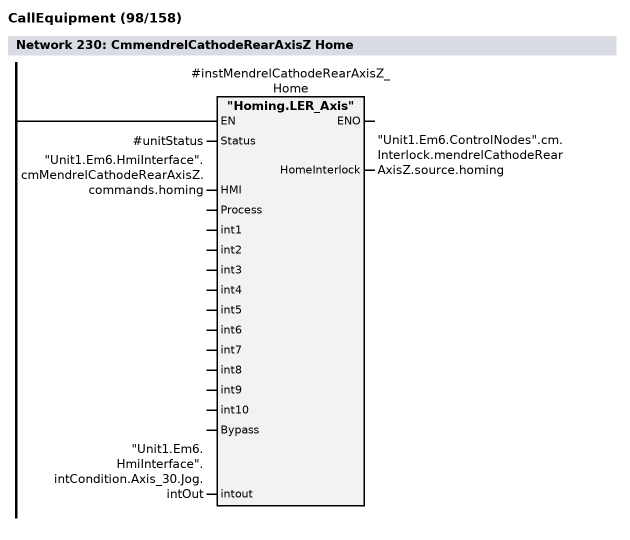
   RUNG wire#powerrail
      #instMendrelCathodeRearAxisZ_Home(Status := #unitStatus, HMI := "Unit1.Em6.HmiInterface".cmMendrelCathodeRearAxisZ.commands.homing, Process :=, int1 :=, int2 :=, int3 :=, int4 :=, int5 :=, int6 :=, int7 :=, int8 :=, int9 :=, int10 :=, Bypass :=, intout := "Unit1.Em6.HmiInterface".intCondition.Axis_30.Jog.intOut, HomeInterlock => "Unit1.Em6.ControlNodes".cm.Interlock.mendrelCathodeRearAxisZ.source.homing)
   END_RUNG
   // the same network as SCL:
   #instMendrelCathodeRearAxisZ_Home(Status := #unitStatus,   // "Homing.LER_Axis"
                           HMI := "Unit1.Em6.HmiInterface".cmMendrelCathodeRearAxisZ.commands.homing,
                           intout := "Unit1.Em6.HmiInterface".intCondition.Axis_30.Jog.intOut,
                           HomeInterlock => "Unit1.Em6.ControlNodes".cm.Interlock.mendrelCathodeRearAxisZ.source.homing);
END_REGION

REGION Network 231: CmmendrelCathodeRearAxisZ Position Absolute Jog
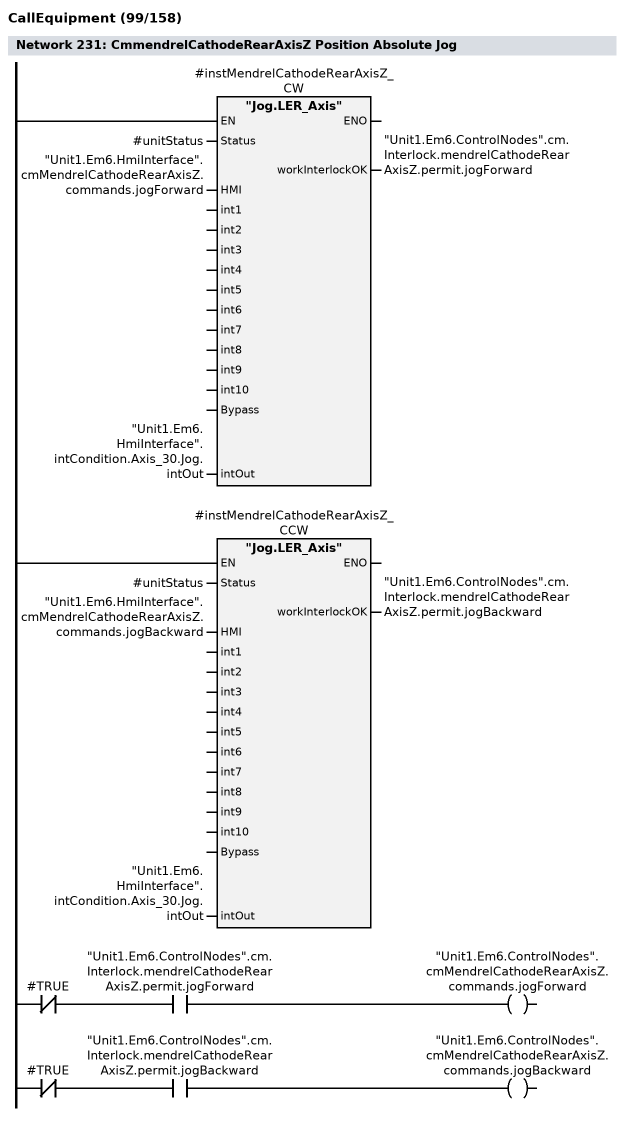
   RUNG wire#powerrail
      #instMendrelCathodeRearAxisZ_CW(Status := #unitStatus, HMI := "Unit1.Em6.HmiInterface".cmMendrelCathodeRearAxisZ.commands.jogForward, int1 :=, int2 :=, int3 :=, int4 :=, int5 :=, int6 :=, int7 :=, int8 :=, int9 :=, int10 :=, Bypass :=, intOut := "Unit1.Em6.HmiInterface".intCondition.Axis_30.Jog.intOut, workInterlockOK => "Unit1.Em6.ControlNodes".cm.Interlock.mendrelCathodeRearAxisZ.permit.jogForward)
   END_RUNG
   RUNG wire#powerrail
      #instMendrelCathodeRearAxisZ_CCW(Status := #unitStatus, HMI := "Unit1.Em6.HmiInterface".cmMendrelCathodeRearAxisZ.commands.jogBackward, int1 :=, int2 :=, int3 :=, int4 :=, int5 :=, int6 :=, int7 :=, int8 :=, int9 :=, int10 :=, Bypass :=, intOut := "Unit1.Em6.HmiInterface".intCondition.Axis_30.Jog.intOut, workInterlockOK => "Unit1.Em6.ControlNodes".cm.Interlock.mendrelCathodeRearAxisZ.permit.jogBackward)
   END_RUNG
   RUNG wire#powerrail
      I_Contact( #TRUE )
      Contact( "Unit1.Em6.ControlNodes".cm.Interlock.mendrelCathodeRearAxisZ.permit.jogForward )
      Coil( "Unit1.Em6.ControlNodes".cmMendrelCathodeRearAxisZ.commands.jogForward )
   END_RUNG
   RUNG wire#powerrail
      I_Contact( #TRUE )
      Contact( "Unit1.Em6.ControlNodes".cm.Interlock.mendrelCathodeRearAxisZ.permit.jogBackward )
      Coil( "Unit1.Em6.ControlNodes".cmMendrelCathodeRearAxisZ.commands.jogBackward )
   END_RUNG
   // the same network as SCL:
   #instMendrelCathodeRearAxisZ_CW(Status := #unitStatus,   // "Jog.LER_Axis"
                           HMI := "Unit1.Em6.HmiInterface".cmMendrelCathodeRearAxisZ.commands.jogForward,
                           intOut := "Unit1.Em6.HmiInterface".intCondition.Axis_30.Jog.intOut,
                           workInterlockOK => "Unit1.Em6.ControlNodes".cm.Interlock.mendrelCathodeRearAxisZ.permit.jogForward);
   #instMendrelCathodeRearAxisZ_CCW(Status := #unitStatus,   // "Jog.LER_Axis"
                           HMI := "Unit1.Em6.HmiInterface".cmMendrelCathodeRearAxisZ.commands.jogBackward,
                           intOut := "Unit1.Em6.HmiInterface".intCondition.Axis_30.Jog.intOut,
                           workInterlockOK => "Unit1.Em6.ControlNodes".cm.Interlock.mendrelCathodeRearAxisZ.permit.jogBackward);
   "Unit1.Em6.ControlNodes".cmMendrelCathodeRearAxisZ.commands.jogForward := NOT #TRUE AND "Unit1.Em6.ControlNodes".cm.Interlock.mendrelCathodeRearAxisZ.permit.jogForward;
   "Unit1.Em6.ControlNodes".cmMendrelCathodeRearAxisZ.commands.jogBackward := NOT #TRUE AND "Unit1.Em6.ControlNodes".cm.Interlock.mendrelCathodeRearAxisZ.permit.jogBackward;
END_REGION

REGION Network 232: CmmendrelCathodeRearAxisZ Position Absolute Position0
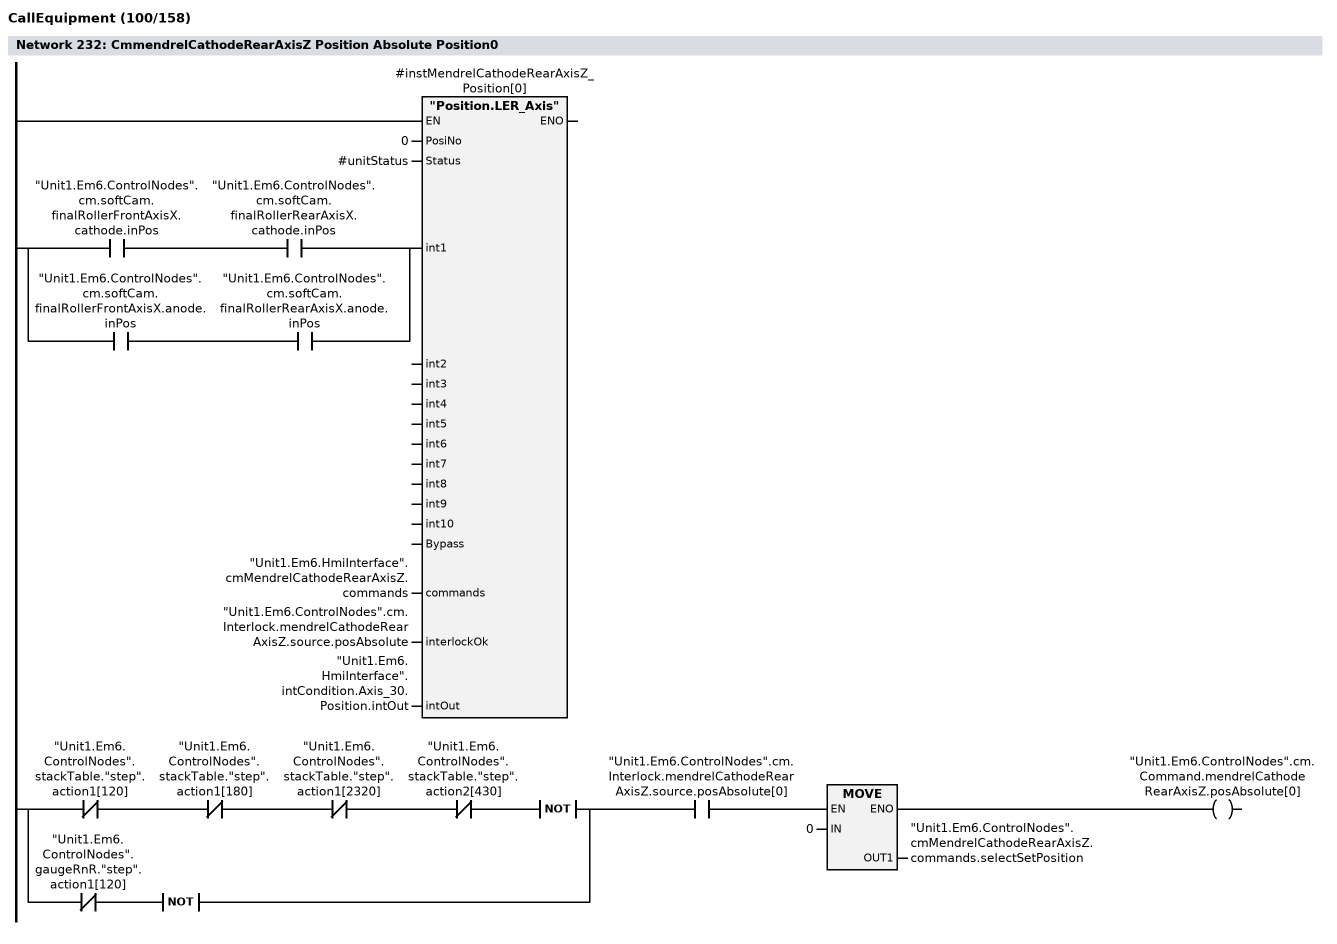
   RUNG wire#powerrail
      #instMendrelCathodeRearAxisZ_Position[0](int1 := wire#w1, PosiNo := 0, Status := #unitStatus, int2 :=, int3 :=, int4 :=, int5 :=, int6 :=, int7 :=, int8 :=, int9 :=, int10 :=, Bypass :=, commands := "Unit1.Em6.HmiInterface".cmMendrelCathodeRearAxisZ.commands, interlockOk := "Unit1.Em6.ControlNodes".cm.Interlock.mendrelCathodeRearAxisZ.source.posAbsolute, intOut := "Unit1.Em6.HmiInterface".intCondition.Axis_30.Position.intOut)
   END_RUNG
   RUNG wire#powerrail
      Contact( "Unit1.Em6.ControlNodes".cm.softCam.finalRollerFrontAxisX.cathode.inPos )
      Contact( "Unit1.Em6.ControlNodes".cm.softCam.finalRollerRearAxisX.cathode.inPos )
   END_RUNG wire#w1
   RUNG wire#powerrail
      Contact( "Unit1.Em6.ControlNodes".cm.softCam.finalRollerFrontAxisX.anode.inPos )
      Contact( "Unit1.Em6.ControlNodes".cm.softCam.finalRollerRearAxisX.anode.inPos )
   END_RUNG wire#w1
   RUNG wire#powerrail
      I_Contact( "Unit1.Em6.ControlNodes".stackTable."step".action1[120] )
      I_Contact( "Unit1.Em6.ControlNodes".stackTable."step".action1[180] )
      I_Contact( "Unit1.Em6.ControlNodes".stackTable."step".action1[2320] )
      I_Contact( "Unit1.Em6.ControlNodes".stackTable."step".action2[430] )
      Not()
      wire#w2
      Contact( "Unit1.Em6.ControlNodes".cm.Interlock.mendrelCathodeRearAxisZ.source.posAbsolute[0] )
      Move(in := 0, out1 => "Unit1.Em6.ControlNodes".cmMendrelCathodeRearAxisZ.commands.selectSetPosition)
      Coil( "Unit1.Em6.ControlNodes".cm.Command.mendrelCathodeRearAxisZ.posAbsolute[0] )
   END_RUNG
   RUNG wire#powerrail
      I_Contact( "Unit1.Em6.ControlNodes".gaugeRnR."step".action1[120] )
      Not()
   END_RUNG wire#w2
   // the same network as SCL:
   #instMendrelCathodeRearAxisZ_Position[0](PosiNo := 0,   // "Position.LER_Axis"
                           Status := #unitStatus,
                           int1 := ("Unit1.Em6.ControlNodes".cm.softCam.finalRollerFrontAxisX.cathode.inPos AND "Unit1.Em6.ControlNodes".cm.softCam.finalRollerRearAxisX.cathode.inPos) OR ("Unit1.Em6.ControlNodes".cm.softCam.finalRollerFrontAxisX.anode.inPos AND "Unit1.Em6.ControlNodes".cm.softCam.finalRollerRearAxisX.anode.inPos),
                           commands := "Unit1.Em6.HmiInterface".cmMendrelCathodeRearAxisZ.commands,
                           interlockOk := "Unit1.Em6.ControlNodes".cm.Interlock.mendrelCathodeRearAxisZ.source.posAbsolute,
                           intOut := "Unit1.Em6.HmiInterface".intCondition.Axis_30.Position.intOut);
   #_w1 := (NOT (NOT "Unit1.Em6.ControlNodes".stackTable."step".action1[120] AND NOT "Unit1.Em6.ControlNodes".stackTable."step".action1[180] AND NOT "Unit1.Em6.ControlNodes".stackTable."step".action1[2320] AND NOT "Unit1.Em6.ControlNodes".stackTable."step".action2[430]) OR NOT (NOT "Unit1.Em6.ControlNodes".gaugeRnR."step".action1[120])) AND "Unit1.Em6.ControlNodes".cm.Interlock.mendrelCathodeRearAxisZ.source.posAbsolute[0];
   IF #_w1 THEN "Unit1.Em6.ControlNodes".cmMendrelCathodeRearAxisZ.commands.selectSetPosition := 0; END_IF;
   "Unit1.Em6.ControlNodes".cm.Command.mendrelCathodeRearAxisZ.posAbsolute[0] := #_w1;
END_REGION

REGION Network 233: CmmendrelCathodeRearAxisZ Position Absolute Position1
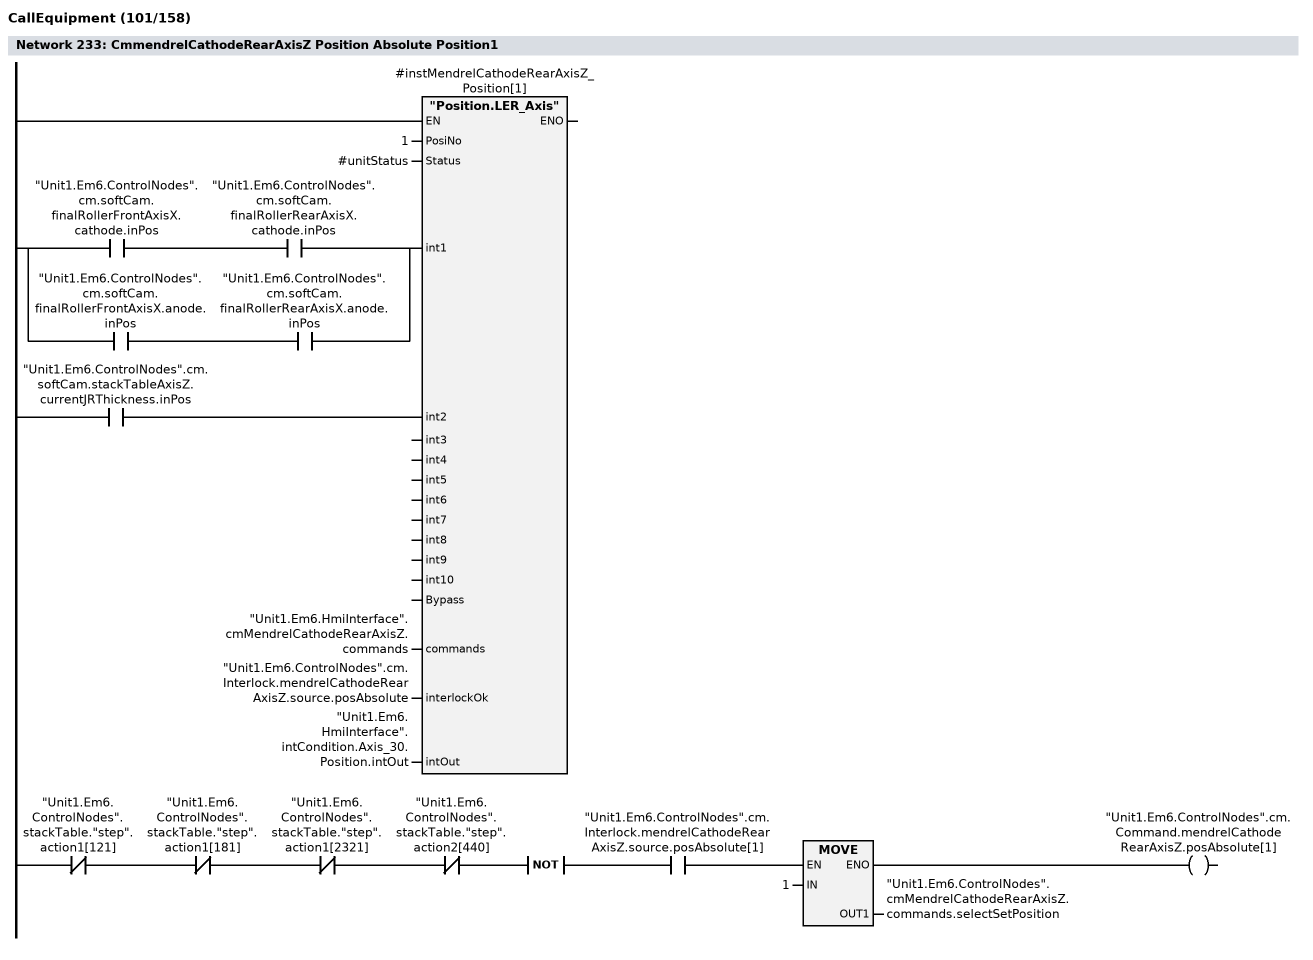
   RUNG wire#powerrail
      #instMendrelCathodeRearAxisZ_Position[1](int1 := wire#w1, int2 := wire#w2, PosiNo := 1, Status := #unitStatus, int3 :=, int4 :=, int5 :=, int6 :=, int7 :=, int8 :=, int9 :=, int10 :=, Bypass :=, commands := "Unit1.Em6.HmiInterface".cmMendrelCathodeRearAxisZ.commands, interlockOk := "Unit1.Em6.ControlNodes".cm.Interlock.mendrelCathodeRearAxisZ.source.posAbsolute, intOut := "Unit1.Em6.HmiInterface".intCondition.Axis_30.Position.intOut)
   END_RUNG
   RUNG wire#powerrail
      Contact( "Unit1.Em6.ControlNodes".cm.softCam.finalRollerFrontAxisX.cathode.inPos )
      Contact( "Unit1.Em6.ControlNodes".cm.softCam.finalRollerRearAxisX.cathode.inPos )
   END_RUNG wire#w1
   RUNG wire#powerrail
      Contact( "Unit1.Em6.ControlNodes".cm.softCam.finalRollerFrontAxisX.anode.inPos )
      Contact( "Unit1.Em6.ControlNodes".cm.softCam.finalRollerRearAxisX.anode.inPos )
   END_RUNG wire#w1
   RUNG wire#powerrail
      Contact( "Unit1.Em6.ControlNodes".cm.softCam.stackTableAxisZ.currentJRThickness.inPos )
   END_RUNG wire#w2
   RUNG wire#powerrail
      I_Contact( "Unit1.Em6.ControlNodes".stackTable."step".action1[121] )
      I_Contact( "Unit1.Em6.ControlNodes".stackTable."step".action1[181] )
      I_Contact( "Unit1.Em6.ControlNodes".stackTable."step".action1[2321] )
      I_Contact( "Unit1.Em6.ControlNodes".stackTable."step".action2[440] )
      Not()
      Contact( "Unit1.Em6.ControlNodes".cm.Interlock.mendrelCathodeRearAxisZ.source.posAbsolute[1] )
      Move(in := 1, out1 => "Unit1.Em6.ControlNodes".cmMendrelCathodeRearAxisZ.commands.selectSetPosition)
      Coil( "Unit1.Em6.ControlNodes".cm.Command.mendrelCathodeRearAxisZ.posAbsolute[1] )
   END_RUNG
   // the same network as SCL:
   #instMendrelCathodeRearAxisZ_Position[1](PosiNo := 1,   // "Position.LER_Axis"
                           Status := #unitStatus,
                           int1 := ("Unit1.Em6.ControlNodes".cm.softCam.finalRollerFrontAxisX.cathode.inPos AND "Unit1.Em6.ControlNodes".cm.softCam.finalRollerRearAxisX.cathode.inPos) OR ("Unit1.Em6.ControlNodes".cm.softCam.finalRollerFrontAxisX.anode.inPos AND "Unit1.Em6.ControlNodes".cm.softCam.finalRollerRearAxisX.anode.inPos),
                           int2 := "Unit1.Em6.ControlNodes".cm.softCam.stackTableAxisZ.currentJRThickness.inPos,
                           commands := "Unit1.Em6.HmiInterface".cmMendrelCathodeRearAxisZ.commands,
                           interlockOk := "Unit1.Em6.ControlNodes".cm.Interlock.mendrelCathodeRearAxisZ.source.posAbsolute,
                           intOut := "Unit1.Em6.HmiInterface".intCondition.Axis_30.Position.intOut);
   #_w1 := NOT (NOT "Unit1.Em6.ControlNodes".stackTable."step".action1[121] AND NOT "Unit1.Em6.ControlNodes".stackTable."step".action1[181] AND NOT "Unit1.Em6.ControlNodes".stackTable."step".action1[2321] AND NOT "Unit1.Em6.ControlNodes".stackTable."step".action2[440]) AND "Unit1.Em6.ControlNodes".cm.Interlock.mendrelCathodeRearAxisZ.source.posAbsolute[1];
   IF #_w1 THEN "Unit1.Em6.ControlNodes".cmMendrelCathodeRearAxisZ.commands.selectSetPosition := 1; END_IF;
   "Unit1.Em6.ControlNodes".cm.Command.mendrelCathodeRearAxisZ.posAbsolute[1] := #_w1;
END_REGION

REGION Network 234: CmmendrelCathodeRearAxisZ Position Absolute Position2
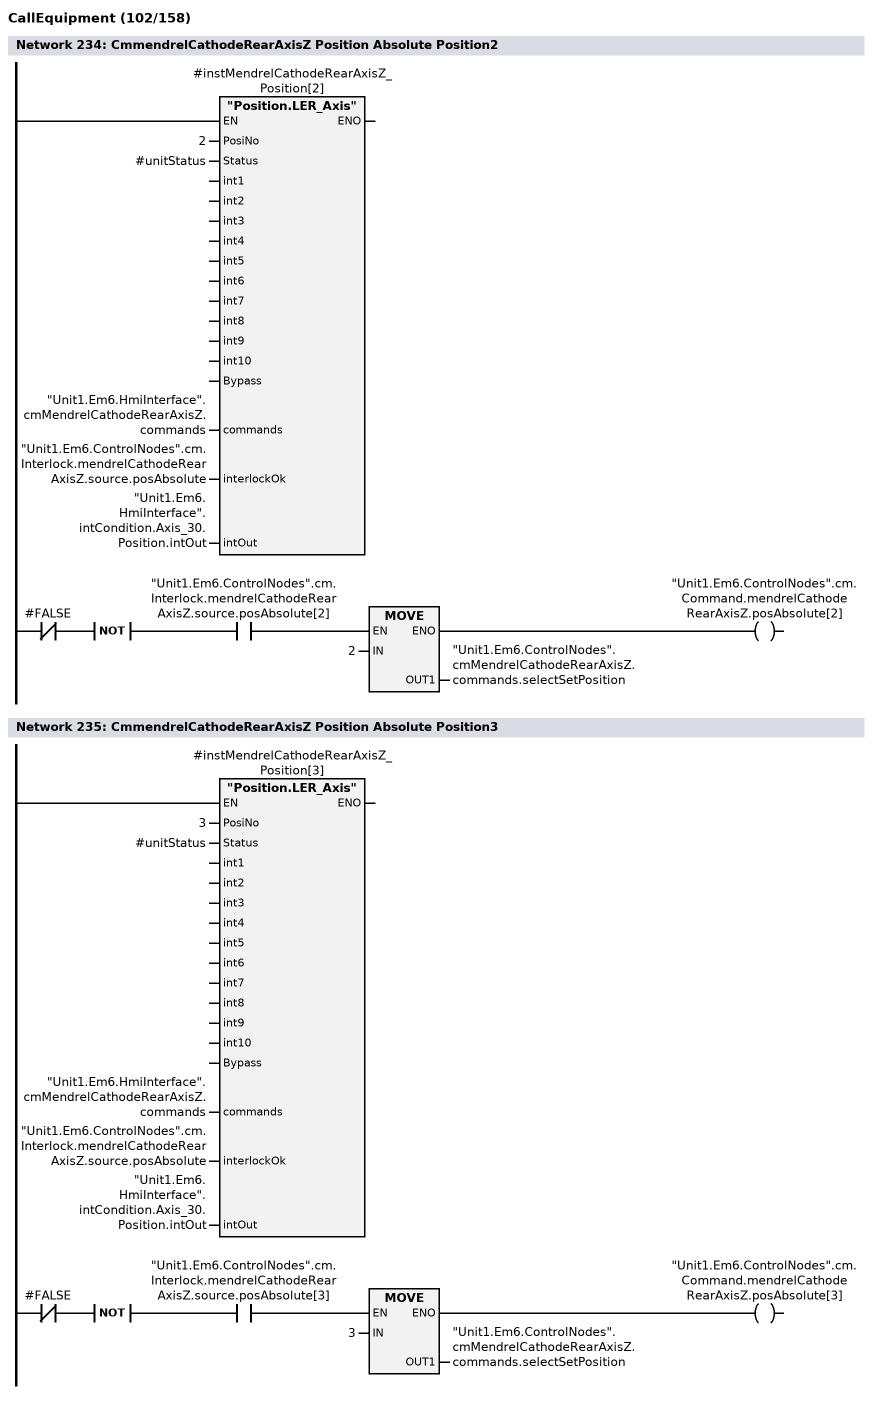
   RUNG wire#powerrail
      #instMendrelCathodeRearAxisZ_Position[2](PosiNo := 2, Status := #unitStatus, int1 :=, int2 :=, int3 :=, int4 :=, int5 :=, int6 :=, int7 :=, int8 :=, int9 :=, int10 :=, Bypass :=, commands := "Unit1.Em6.HmiInterface".cmMendrelCathodeRearAxisZ.commands, interlockOk := "Unit1.Em6.ControlNodes".cm.Interlock.mendrelCathodeRearAxisZ.source.posAbsolute, intOut := "Unit1.Em6.HmiInterface".intCondition.Axis_30.Position.intOut)
   END_RUNG
   RUNG wire#powerrail
      I_Contact( #FALSE )
      Not()
      Contact( "Unit1.Em6.ControlNodes".cm.Interlock.mendrelCathodeRearAxisZ.source.posAbsolute[2] )
      Move(in := 2, out1 => "Unit1.Em6.ControlNodes".cmMendrelCathodeRearAxisZ.commands.selectSetPosition)
      Coil( "Unit1.Em6.ControlNodes".cm.Command.mendrelCathodeRearAxisZ.posAbsolute[2] )
   END_RUNG
   // the same network as SCL:
   #instMendrelCathodeRearAxisZ_Position[2](PosiNo := 2,   // "Position.LER_Axis"
                           Status := #unitStatus,
                           commands := "Unit1.Em6.HmiInterface".cmMendrelCathodeRearAxisZ.commands,
                           interlockOk := "Unit1.Em6.ControlNodes".cm.Interlock.mendrelCathodeRearAxisZ.source.posAbsolute,
                           intOut := "Unit1.Em6.HmiInterface".intCondition.Axis_30.Position.intOut);
   #_w1 := NOT (NOT #FALSE) AND "Unit1.Em6.ControlNodes".cm.Interlock.mendrelCathodeRearAxisZ.source.posAbsolute[2];
   IF #_w1 THEN "Unit1.Em6.ControlNodes".cmMendrelCathodeRearAxisZ.commands.selectSetPosition := 2; END_IF;
   "Unit1.Em6.ControlNodes".cm.Command.mendrelCathodeRearAxisZ.posAbsolute[2] := #_w1;
END_REGION

REGION Network 235: CmmendrelCathodeRearAxisZ Position Absolute Position3
   RUNG wire#powerrail
      #instMendrelCathodeRearAxisZ_Position[3](PosiNo := 3, Status := #unitStatus, int1 :=, int2 :=, int3 :=, int4 :=, int5 :=, int6 :=, int7 :=, int8 :=, int9 :=, int10 :=, Bypass :=, commands := "Unit1.Em6.HmiInterface".cmMendrelCathodeRearAxisZ.commands, interlockOk := "Unit1.Em6.ControlNodes".cm.Interlock.mendrelCathodeRearAxisZ.source.posAbsolute, intOut := "Unit1.Em6.HmiInterface".intCondition.Axis_30.Position.intOut)
   END_RUNG
   RUNG wire#powerrail
      I_Contact( #FALSE )
      Not()
      Contact( "Unit1.Em6.ControlNodes".cm.Interlock.mendrelCathodeRearAxisZ.source.posAbsolute[3] )
      Move(in := 3, out1 => "Unit1.Em6.ControlNodes".cmMendrelCathodeRearAxisZ.commands.selectSetPosition)
      Coil( "Unit1.Em6.ControlNodes".cm.Command.mendrelCathodeRearAxisZ.posAbsolute[3] )
   END_RUNG
   // the same network as SCL:
   #instMendrelCathodeRearAxisZ_Position[3](PosiNo := 3,   // "Position.LER_Axis"
                           Status := #unitStatus,
                           commands := "Unit1.Em6.HmiInterface".cmMendrelCathodeRearAxisZ.commands,
                           interlockOk := "Unit1.Em6.ControlNodes".cm.Interlock.mendrelCathodeRearAxisZ.source.posAbsolute,
                           intOut := "Unit1.Em6.HmiInterface".intCondition.Axis_30.Position.intOut);
   #_w1 := NOT (NOT #FALSE) AND "Unit1.Em6.ControlNodes".cm.Interlock.mendrelCathodeRearAxisZ.source.posAbsolute[3];
   IF #_w1 THEN "Unit1.Em6.ControlNodes".cmMendrelCathodeRearAxisZ.commands.selectSetPosition := 3; END_IF;
   "Unit1.Em6.ControlNodes".cm.Command.mendrelCathodeRearAxisZ.posAbsolute[3] := #_w1;
END_REGION

REGION Network 236: CmmendrelCathodeRearAxisZ Position Absolute Position4
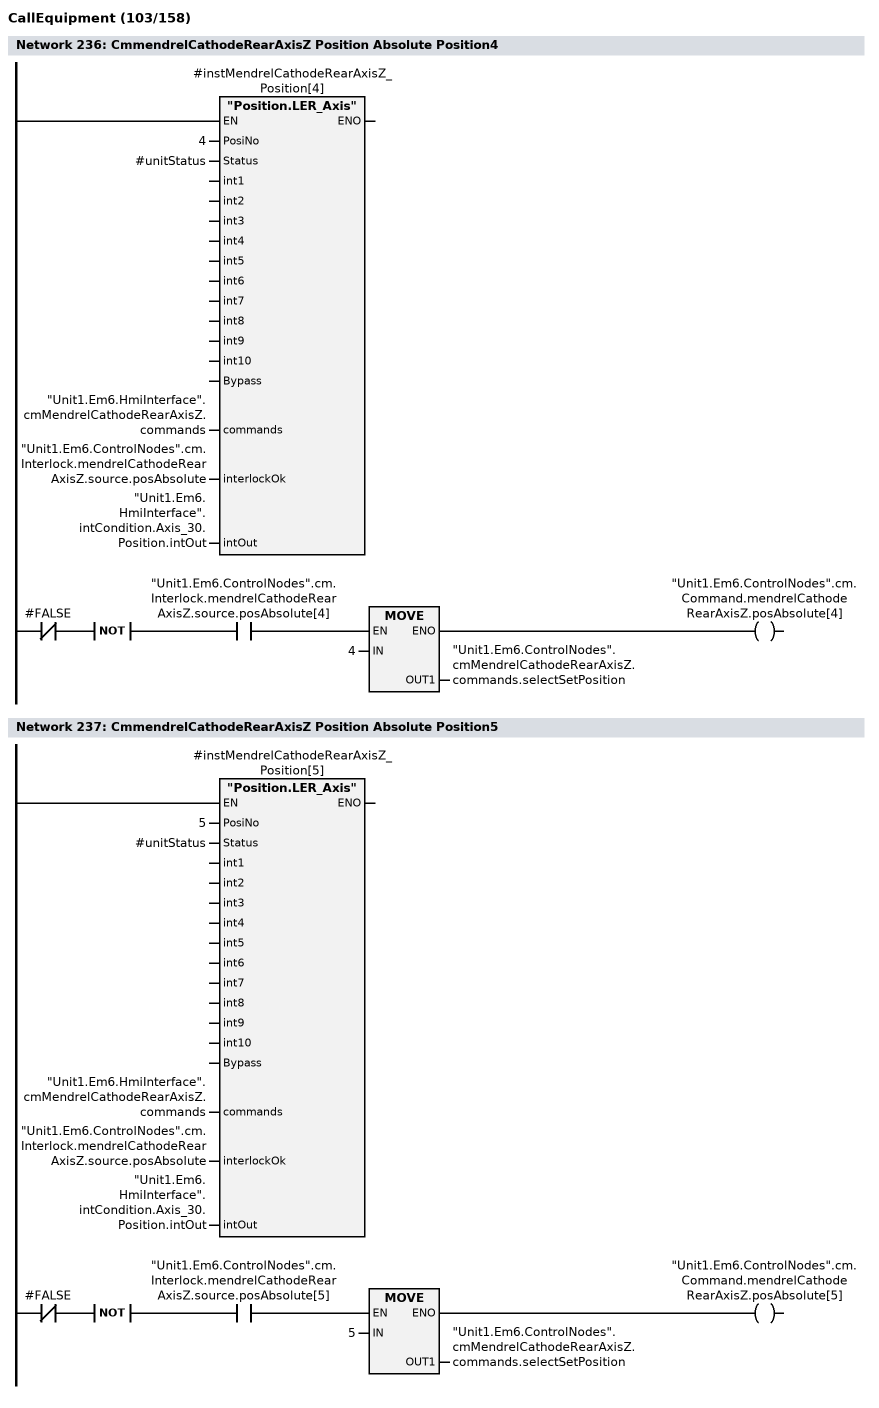
   RUNG wire#powerrail
      #instMendrelCathodeRearAxisZ_Position[4](PosiNo := 4, Status := #unitStatus, int1 :=, int2 :=, int3 :=, int4 :=, int5 :=, int6 :=, int7 :=, int8 :=, int9 :=, int10 :=, Bypass :=, commands := "Unit1.Em6.HmiInterface".cmMendrelCathodeRearAxisZ.commands, interlockOk := "Unit1.Em6.ControlNodes".cm.Interlock.mendrelCathodeRearAxisZ.source.posAbsolute, intOut := "Unit1.Em6.HmiInterface".intCondition.Axis_30.Position.intOut)
   END_RUNG
   RUNG wire#powerrail
      I_Contact( #FALSE )
      Not()
      Contact( "Unit1.Em6.ControlNodes".cm.Interlock.mendrelCathodeRearAxisZ.source.posAbsolute[4] )
      Move(in := 4, out1 => "Unit1.Em6.ControlNodes".cmMendrelCathodeRearAxisZ.commands.selectSetPosition)
      Coil( "Unit1.Em6.ControlNodes".cm.Command.mendrelCathodeRearAxisZ.posAbsolute[4] )
   END_RUNG
   // the same network as SCL:
   #instMendrelCathodeRearAxisZ_Position[4](PosiNo := 4,   // "Position.LER_Axis"
                           Status := #unitStatus,
                           commands := "Unit1.Em6.HmiInterface".cmMendrelCathodeRearAxisZ.commands,
                           interlockOk := "Unit1.Em6.ControlNodes".cm.Interlock.mendrelCathodeRearAxisZ.source.posAbsolute,
                           intOut := "Unit1.Em6.HmiInterface".intCondition.Axis_30.Position.intOut);
   #_w1 := NOT (NOT #FALSE) AND "Unit1.Em6.ControlNodes".cm.Interlock.mendrelCathodeRearAxisZ.source.posAbsolute[4];
   IF #_w1 THEN "Unit1.Em6.ControlNodes".cmMendrelCathodeRearAxisZ.commands.selectSetPosition := 4; END_IF;
   "Unit1.Em6.ControlNodes".cm.Command.mendrelCathodeRearAxisZ.posAbsolute[4] := #_w1;
END_REGION

REGION Network 237: CmmendrelCathodeRearAxisZ Position Absolute Position5
   RUNG wire#powerrail
      #instMendrelCathodeRearAxisZ_Position[5](PosiNo := 5, Status := #unitStatus, int1 :=, int2 :=, int3 :=, int4 :=, int5 :=, int6 :=, int7 :=, int8 :=, int9 :=, int10 :=, Bypass :=, commands := "Unit1.Em6.HmiInterface".cmMendrelCathodeRearAxisZ.commands, interlockOk := "Unit1.Em6.ControlNodes".cm.Interlock.mendrelCathodeRearAxisZ.source.posAbsolute, intOut := "Unit1.Em6.HmiInterface".intCondition.Axis_30.Position.intOut)
   END_RUNG
   RUNG wire#powerrail
      I_Contact( #FALSE )
      Not()
      Contact( "Unit1.Em6.ControlNodes".cm.Interlock.mendrelCathodeRearAxisZ.source.posAbsolute[5] )
      Move(in := 5, out1 => "Unit1.Em6.ControlNodes".cmMendrelCathodeRearAxisZ.commands.selectSetPosition)
      Coil( "Unit1.Em6.ControlNodes".cm.Command.mendrelCathodeRearAxisZ.posAbsolute[5] )
   END_RUNG
   // the same network as SCL:
   #instMendrelCathodeRearAxisZ_Position[5](PosiNo := 5,   // "Position.LER_Axis"
                           Status := #unitStatus,
                           commands := "Unit1.Em6.HmiInterface".cmMendrelCathodeRearAxisZ.commands,
                           interlockOk := "Unit1.Em6.ControlNodes".cm.Interlock.mendrelCathodeRearAxisZ.source.posAbsolute,
                           intOut := "Unit1.Em6.HmiInterface".intCondition.Axis_30.Position.intOut);
   #_w1 := NOT (NOT #FALSE) AND "Unit1.Em6.ControlNodes".cm.Interlock.mendrelCathodeRearAxisZ.source.posAbsolute[5];
   IF #_w1 THEN "Unit1.Em6.ControlNodes".cmMendrelCathodeRearAxisZ.commands.selectSetPosition := 5; END_IF;
   "Unit1.Em6.ControlNodes".cm.Command.mendrelCathodeRearAxisZ.posAbsolute[5] := #_w1;
END_REGION

REGION Network 238: CmmendrelCathodeRearAxisZ Summary Command
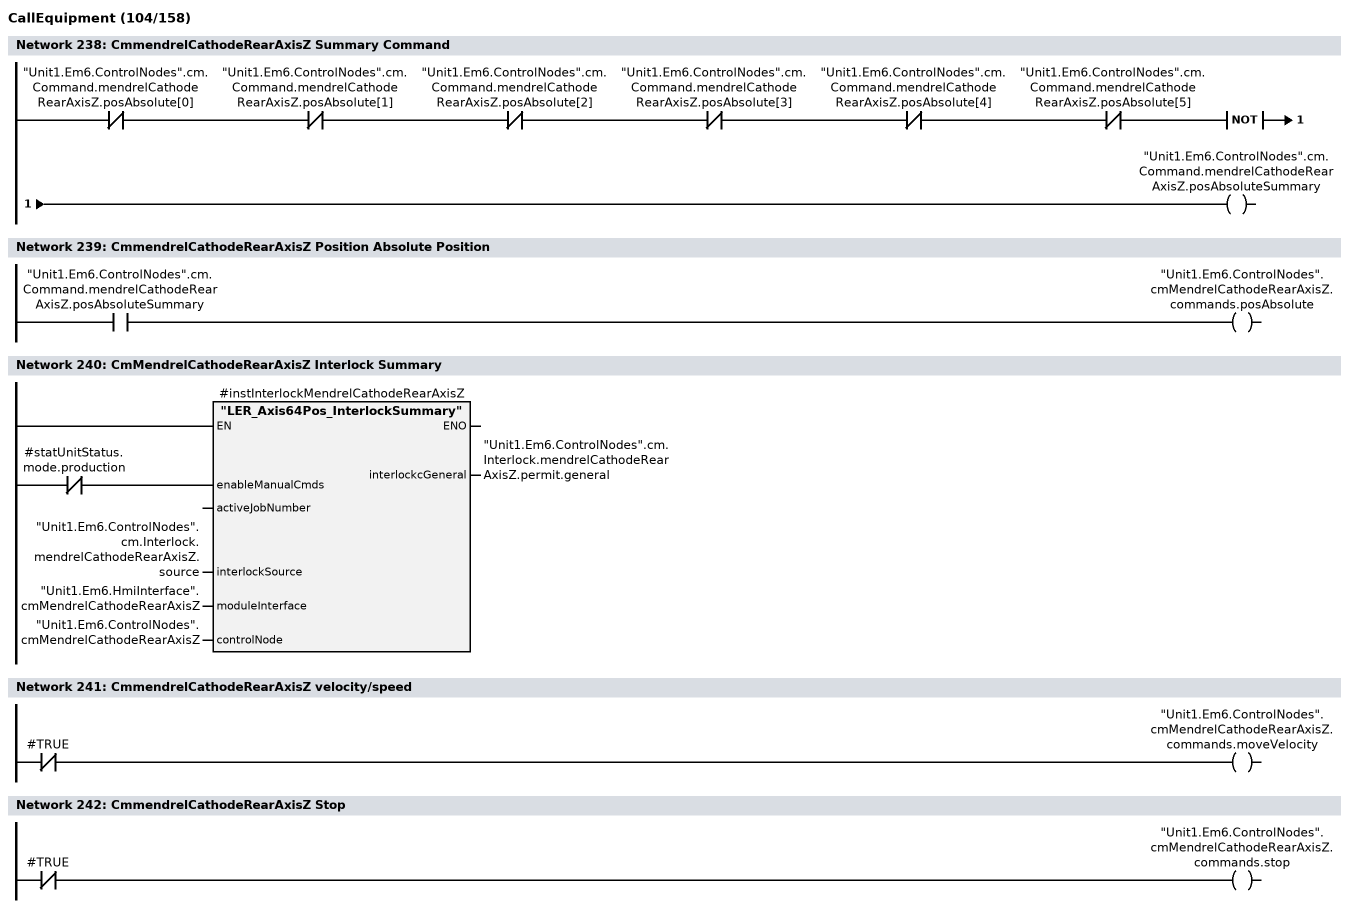
   RUNG wire#powerrail
      I_Contact( "Unit1.Em6.ControlNodes".cm.Command.mendrelCathodeRearAxisZ.posAbsolute[0] )
      I_Contact( "Unit1.Em6.ControlNodes".cm.Command.mendrelCathodeRearAxisZ.posAbsolute[1] )
      I_Contact( "Unit1.Em6.ControlNodes".cm.Command.mendrelCathodeRearAxisZ.posAbsolute[2] )
      I_Contact( "Unit1.Em6.ControlNodes".cm.Command.mendrelCathodeRearAxisZ.posAbsolute[3] )
      I_Contact( "Unit1.Em6.ControlNodes".cm.Command.mendrelCathodeRearAxisZ.posAbsolute[4] )
      I_Contact( "Unit1.Em6.ControlNodes".cm.Command.mendrelCathodeRearAxisZ.posAbsolute[5] )
      Not()
      Coil( "Unit1.Em6.ControlNodes".cm.Command.mendrelCathodeRearAxisZ.posAbsoluteSummary )
   END_RUNG
   // the same network as SCL:
   "Unit1.Em6.ControlNodes".cm.Command.mendrelCathodeRearAxisZ.posAbsoluteSummary := NOT (NOT "Unit1.Em6.ControlNodes".cm.Command.mendrelCathodeRearAxisZ.posAbsolute[0] AND NOT "Unit1.Em6.ControlNodes".cm.Command.mendrelCathodeRearAxisZ.posAbsolute[1] AND NOT "Unit1.Em6.ControlNodes".cm.Command.mendrelCathodeRearAxisZ.posAbsolute[2] AND NOT "Unit1.Em6.ControlNodes".cm.Command.mendrelCathodeRearAxisZ.posAbsolute[3] AND NOT "Unit1.Em6.ControlNodes".cm.Command.mendrelCathodeRearAxisZ.posAbsolute[4] AND NOT "Unit1.Em6.ControlNodes".cm.Command.mendrelCathodeRearAxisZ.posAbsolute[5]);
END_REGION

REGION Network 239: CmmendrelCathodeRearAxisZ Position Absolute Position
   RUNG wire#powerrail
      Contact( "Unit1.Em6.ControlNodes".cm.Command.mendrelCathodeRearAxisZ.posAbsoluteSummary )
      Coil( "Unit1.Em6.ControlNodes".cmMendrelCathodeRearAxisZ.commands.posAbsolute )
   END_RUNG
   // the same network as SCL:
   "Unit1.Em6.ControlNodes".cmMendrelCathodeRearAxisZ.commands.posAbsolute := "Unit1.Em6.ControlNodes".cm.Command.mendrelCathodeRearAxisZ.posAbsoluteSummary;
END_REGION

REGION Network 240: CmMendrelCathodeRearAxisZ Interlock Summary
   RUNG wire#powerrail
      #instInterlockMendrelCathodeRearAxisZ(enableManualCmds := wire#w1, activeJobNumber :=, interlockSource := "Unit1.Em6.ControlNodes".cm.Interlock.mendrelCathodeRearAxisZ.source, moduleInterface := "Unit1.Em6.HmiInterface".cmMendrelCathodeRearAxisZ, controlNode := "Unit1.Em6.ControlNodes".cmMendrelCathodeRearAxisZ, interlockcGeneral => "Unit1.Em6.ControlNodes".cm.Interlock.mendrelCathodeRearAxisZ.permit.general)
   END_RUNG
   RUNG wire#powerrail
      I_Contact( #statUnitStatus.mode.production )
   END_RUNG wire#w1
   // the same network as SCL:
   #instInterlockMendrelCathodeRearAxisZ(enableManualCmds := NOT #statUnitStatus.mode.production,   // "LER_Axis64Pos_InterlockSummary"
                           interlockSource := "Unit1.Em6.ControlNodes".cm.Interlock.mendrelCathodeRearAxisZ.source,
                           moduleInterface := "Unit1.Em6.HmiInterface".cmMendrelCathodeRearAxisZ,
                           controlNode := "Unit1.Em6.ControlNodes".cmMendrelCathodeRearAxisZ,
                           interlockcGeneral => "Unit1.Em6.ControlNodes".cm.Interlock.mendrelCathodeRearAxisZ.permit.general);
END_REGION

REGION Network 241: CmmendrelCathodeRearAxisZ velocity/speed
   RUNG wire#powerrail
      I_Contact( #TRUE )
      Coil( "Unit1.Em6.ControlNodes".cmMendrelCathodeRearAxisZ.commands.moveVelocity )
   END_RUNG
   // the same network as SCL:
   "Unit1.Em6.ControlNodes".cmMendrelCathodeRearAxisZ.commands.moveVelocity := NOT #TRUE;
END_REGION

REGION Network 242: CmmendrelCathodeRearAxisZ Stop
   RUNG wire#powerrail
      I_Contact( #TRUE )
      Coil( "Unit1.Em6.ControlNodes".cmMendrelCathodeRearAxisZ.commands.stop )
   END_RUNG
   // the same network as SCL:
   "Unit1.Em6.ControlNodes".cmMendrelCathodeRearAxisZ.commands.stop := NOT #TRUE;
END_REGION

REGION Network 243: Call CM Cathode Mandrel Rear Z-Axis (LBC_Axis64Pos)
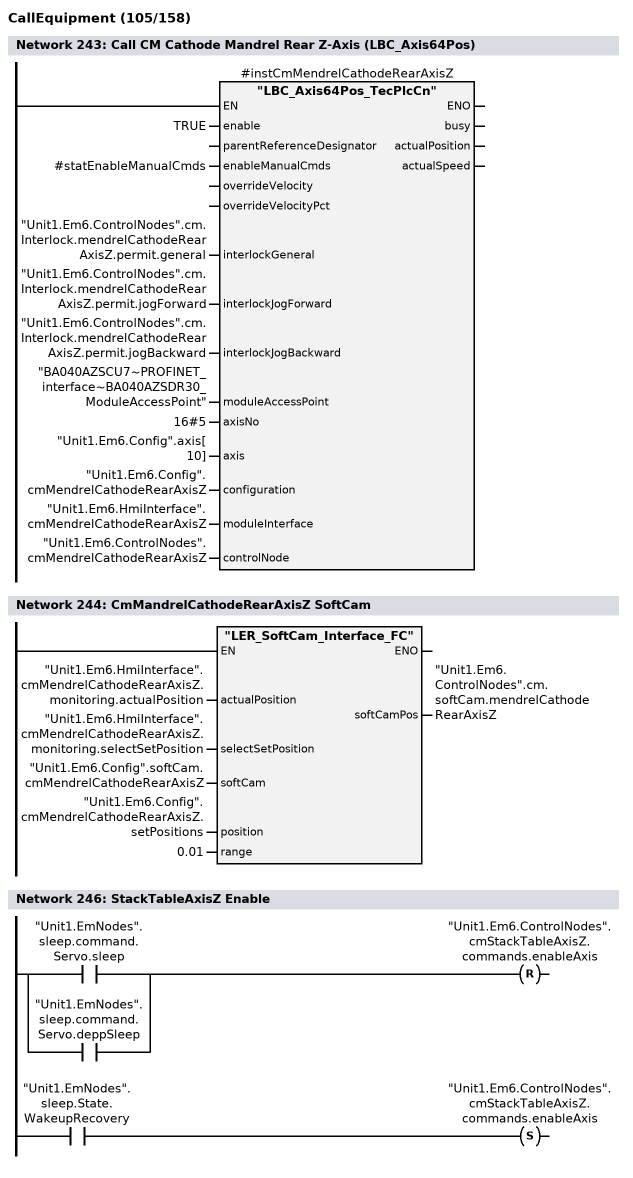
   RUNG wire#powerrail
      #instCmMendrelCathodeRearAxisZ(enable := TRUE, parentReferenceDesignator :=, enableManualCmds := #statEnableManualCmds, overrideVelocity :=, overrideVelocityPct :=, interlockGeneral := "Unit1.Em6.ControlNodes".cm.Interlock.mendrelCathodeRearAxisZ.permit.general, interlockJogForward := "Unit1.Em6.ControlNodes".cm.Interlock.mendrelCathodeRearAxisZ.permit.jogForward, interlockJogBackward := "Unit1.Em6.ControlNodes".cm.Interlock.mendrelCathodeRearAxisZ.permit.jogBackward, moduleAccessPoint := "BA040AZSCU7~PROFINET_interface~BA040AZSDR30_ModuleAccessPoint", axisNo := 16#5, axis := "Unit1.Em6.Config".axis[10], configuration := "Unit1.Em6.Config".cmMendrelCathodeRearAxisZ, moduleInterface := "Unit1.Em6.HmiInterface".cmMendrelCathodeRearAxisZ, controlNode := "Unit1.Em6.ControlNodes".cmMendrelCathodeRearAxisZ, busy =>, actualPosition =>, actualSpeed =>)
   END_RUNG
   // the same network as SCL:
   #instCmMendrelCathodeRearAxisZ(enable := TRUE,   // "LBC_Axis64Pos_TecPlcCn"
                           enableManualCmds := #statEnableManualCmds,
                           interlockGeneral := "Unit1.Em6.ControlNodes".cm.Interlock.mendrelCathodeRearAxisZ.permit.general,
                           interlockJogForward := "Unit1.Em6.ControlNodes".cm.Interlock.mendrelCathodeRearAxisZ.permit.jogForward,
                           interlockJogBackward := "Unit1.Em6.ControlNodes".cm.Interlock.mendrelCathodeRearAxisZ.permit.jogBackward,
                           moduleAccessPoint := "BA040AZSCU7~PROFINET_interface~BA040AZSDR30_ModuleAccessPoint",
                           axisNo := 16#5,
                           axis := "Unit1.Em6.Config".axis[10],
                           configuration := "Unit1.Em6.Config".cmMendrelCathodeRearAxisZ,
                           moduleInterface := "Unit1.Em6.HmiInterface".cmMendrelCathodeRearAxisZ,
                           controlNode := "Unit1.Em6.ControlNodes".cmMendrelCathodeRearAxisZ);
END_REGION

REGION Network 244: CmMandrelCathodeRearAxisZ SoftCam
   RUNG wire#powerrail
      "LER_SoftCam_Interface_FC"(actualPosition := "Unit1.Em6.HmiInterface".cmMendrelCathodeRearAxisZ.monitoring.actualPosition, selectSetPosition := "Unit1.Em6.HmiInterface".cmMendrelCathodeRearAxisZ.monitoring.selectSetPosition, softCam := "Unit1.Em6.Config".softCam.cmMendrelCathodeRearAxisZ, position := "Unit1.Em6.Config".cmMendrelCathodeRearAxisZ.setPositions, range := 0.01, softCamPos => "Unit1.Em6.ControlNodes".cm.softCam.mendrelCathodeRearAxisZ)
   END_RUNG
   // the same network as SCL:
   "LER_SoftCam_Interface_FC"(actualPosition := "Unit1.Em6.HmiInterface".cmMendrelCathodeRearAxisZ.monitoring.actualPosition,
                           selectSetPosition := "Unit1.Em6.HmiInterface".cmMendrelCathodeRearAxisZ.monitoring.selectSetPosition,
                           softCam := "Unit1.Em6.Config".softCam.cmMendrelCathodeRearAxisZ,
                           position := "Unit1.Em6.Config".cmMendrelCathodeRearAxisZ.setPositions,
                           range := 0.01,
                           softCamPos => "Unit1.Em6.ControlNodes".cm.softCam.mendrelCathodeRearAxisZ);
END_REGION

REGION Network 246: StackTableAxisZ Enable
   RUNG wire#powerrail
      Contact( "Unit1.EmNodes".sleep.command.Servo.sleep )
      wire#w1
      R_Coil( "Unit1.Em6.ControlNodes".cmStackTableAxisZ.commands.enableAxis )
   END_RUNG
   RUNG wire#powerrail
      Contact( "Unit1.EmNodes".sleep.command.Servo.deppSleep )
   END_RUNG wire#w1
   RUNG wire#powerrail
      Contact( "Unit1.EmNodes".sleep.State.WakeupRecovery )
      S_Coil( "Unit1.Em6.ControlNodes".cmStackTableAxisZ.commands.enableAxis )
   END_RUNG
   // the same network as SCL:
   IF "Unit1.EmNodes".sleep.command.Servo.sleep OR "Unit1.EmNodes".sleep.command.Servo.deppSleep THEN
       "Unit1.Em6.ControlNodes".cmStackTableAxisZ.commands.enableAxis := FALSE;
   END_IF;
   IF "Unit1.EmNodes".sleep.State.WakeupRecovery THEN
       "Unit1.Em6.ControlNodes".cmStackTableAxisZ.commands.enableAxis := TRUE;
   END_IF;
END_REGION

REGION Network 247: CmStackTableAxisZ Home
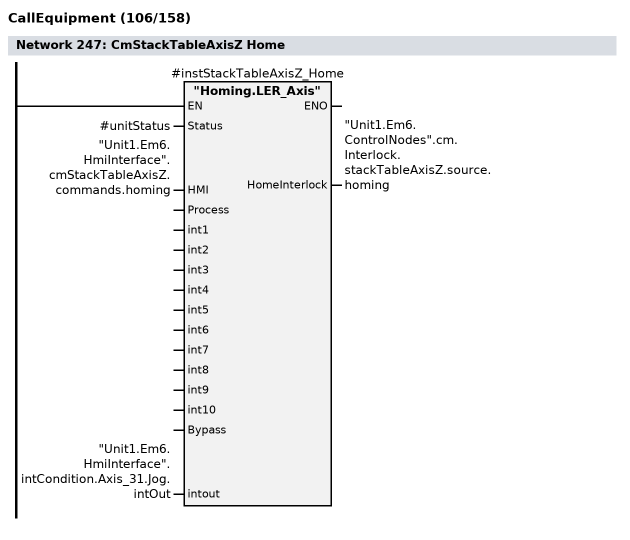
   RUNG wire#powerrail
      #instStackTableAxisZ_Home(Status := #unitStatus, HMI := "Unit1.Em6.HmiInterface".cmStackTableAxisZ.commands.homing, Process :=, int1 :=, int2 :=, int3 :=, int4 :=, int5 :=, int6 :=, int7 :=, int8 :=, int9 :=, int10 :=, Bypass :=, intout := "Unit1.Em6.HmiInterface".intCondition.Axis_31.Jog.intOut, HomeInterlock => "Unit1.Em6.ControlNodes".cm.Interlock.stackTableAxisZ.source.homing)
   END_RUNG
   // the same network as SCL:
   #instStackTableAxisZ_Home(Status := #unitStatus,   // "Homing.LER_Axis"
                           HMI := "Unit1.Em6.HmiInterface".cmStackTableAxisZ.commands.homing,
                           intout := "Unit1.Em6.HmiInterface".intCondition.Axis_31.Jog.intOut,
                           HomeInterlock => "Unit1.Em6.ControlNodes".cm.Interlock.stackTableAxisZ.source.homing);
END_REGION

REGION Network 248: CmStackTableAxisZ Position Absolute Jog
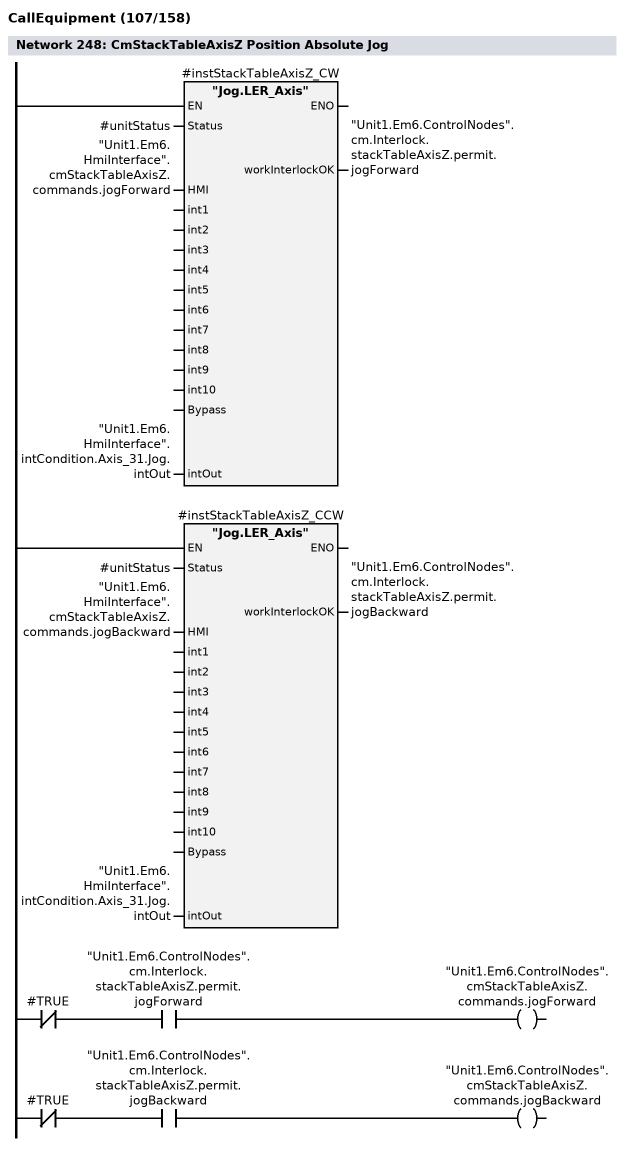
   RUNG wire#powerrail
      #instStackTableAxisZ_CW(Status := #unitStatus, HMI := "Unit1.Em6.HmiInterface".cmStackTableAxisZ.commands.jogForward, int1 :=, int2 :=, int3 :=, int4 :=, int5 :=, int6 :=, int7 :=, int8 :=, int9 :=, int10 :=, Bypass :=, intOut := "Unit1.Em6.HmiInterface".intCondition.Axis_31.Jog.intOut, workInterlockOK => "Unit1.Em6.ControlNodes".cm.Interlock.stackTableAxisZ.permit.jogForward)
   END_RUNG
   RUNG wire#powerrail
      #instStackTableAxisZ_CCW(Status := #unitStatus, HMI := "Unit1.Em6.HmiInterface".cmStackTableAxisZ.commands.jogBackward, int1 :=, int2 :=, int3 :=, int4 :=, int5 :=, int6 :=, int7 :=, int8 :=, int9 :=, int10 :=, Bypass :=, intOut := "Unit1.Em6.HmiInterface".intCondition.Axis_31.Jog.intOut, workInterlockOK => "Unit1.Em6.ControlNodes".cm.Interlock.stackTableAxisZ.permit.jogBackward)
   END_RUNG
   RUNG wire#powerrail
      I_Contact( #TRUE )
      Contact( "Unit1.Em6.ControlNodes".cm.Interlock.stackTableAxisZ.permit.jogForward )
      Coil( "Unit1.Em6.ControlNodes".cmStackTableAxisZ.commands.jogForward )
   END_RUNG
   RUNG wire#powerrail
      I_Contact( #TRUE )
      Contact( "Unit1.Em6.ControlNodes".cm.Interlock.stackTableAxisZ.permit.jogBackward )
      Coil( "Unit1.Em6.ControlNodes".cmStackTableAxisZ.commands.jogBackward )
   END_RUNG
   // the same network as SCL:
   #instStackTableAxisZ_CW(Status := #unitStatus,   // "Jog.LER_Axis"
                           HMI := "Unit1.Em6.HmiInterface".cmStackTableAxisZ.commands.jogForward,
                           intOut := "Unit1.Em6.HmiInterface".intCondition.Axis_31.Jog.intOut,
                           workInterlockOK => "Unit1.Em6.ControlNodes".cm.Interlock.stackTableAxisZ.permit.jogForward);
   #instStackTableAxisZ_CCW(Status := #unitStatus,   // "Jog.LER_Axis"
                           HMI := "Unit1.Em6.HmiInterface".cmStackTableAxisZ.commands.jogBackward,
                           intOut := "Unit1.Em6.HmiInterface".intCondition.Axis_31.Jog.intOut,
                           workInterlockOK => "Unit1.Em6.ControlNodes".cm.Interlock.stackTableAxisZ.permit.jogBackward);
   "Unit1.Em6.ControlNodes".cmStackTableAxisZ.commands.jogForward := NOT #TRUE AND "Unit1.Em6.ControlNodes".cm.Interlock.stackTableAxisZ.permit.jogForward;
   "Unit1.Em6.ControlNodes".cmStackTableAxisZ.commands.jogBackward := NOT #TRUE AND "Unit1.Em6.ControlNodes".cm.Interlock.stackTableAxisZ.permit.jogBackward;
END_REGION

REGION Network 249: CmStackTableAxisZ Position Absolute Position0
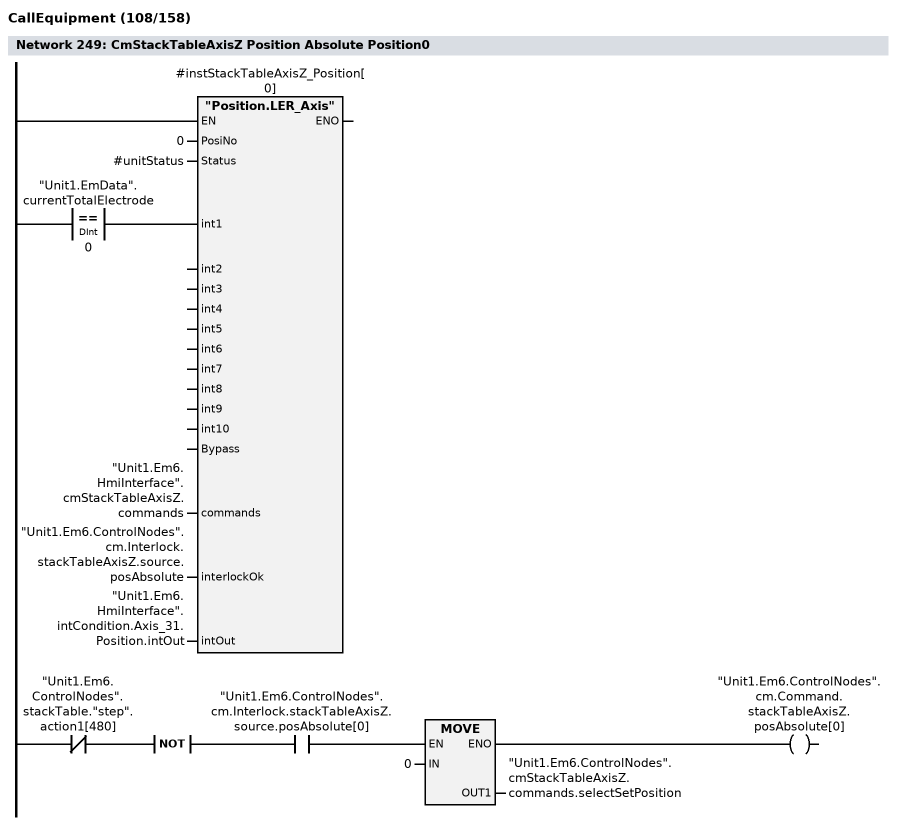
   RUNG wire#powerrail
      #instStackTableAxisZ_Position[0](int1 := wire#w1, PosiNo := 0, Status := #unitStatus, int2 :=, int3 :=, int4 :=, int5 :=, int6 :=, int7 :=, int8 :=, int9 :=, int10 :=, Bypass :=, commands := "Unit1.Em6.HmiInterface".cmStackTableAxisZ.commands, interlockOk := "Unit1.Em6.ControlNodes".cm.Interlock.stackTableAxisZ.source.posAbsolute, intOut := "Unit1.Em6.HmiInterface".intCondition.Axis_31.Position.intOut)
   END_RUNG
   RUNG wire#powerrail
      { S7_Templates := "SrcType := DInt" } EQ_Contact(in1 := "Unit1.EmData".currentTotalElectrode, in2 := 0)
   END_RUNG wire#w1
   RUNG wire#powerrail
      I_Contact( "Unit1.Em6.ControlNodes".stackTable."step".action1[480] )
      Not()
      Contact( "Unit1.Em6.ControlNodes".cm.Interlock.stackTableAxisZ.source.posAbsolute[0] )
      Move(in := 0, out1 => "Unit1.Em6.ControlNodes".cmStackTableAxisZ.commands.selectSetPosition)
      Coil( "Unit1.Em6.ControlNodes".cm.Command.stackTableAxisZ.posAbsolute[0] )
   END_RUNG
   // the same network as SCL:
   #instStackTableAxisZ_Position[0](PosiNo := 0,   // "Position.LER_Axis"
                           Status := #unitStatus,
                           int1 := "Unit1.EmData".currentTotalElectrode = 0,
                           commands := "Unit1.Em6.HmiInterface".cmStackTableAxisZ.commands,
                           interlockOk := "Unit1.Em6.ControlNodes".cm.Interlock.stackTableAxisZ.source.posAbsolute,
                           intOut := "Unit1.Em6.HmiInterface".intCondition.Axis_31.Position.intOut);
   #_w1 := NOT (NOT "Unit1.Em6.ControlNodes".stackTable."step".action1[480]) AND "Unit1.Em6.ControlNodes".cm.Interlock.stackTableAxisZ.source.posAbsolute[0];
   IF #_w1 THEN "Unit1.Em6.ControlNodes".cmStackTableAxisZ.commands.selectSetPosition := 0; END_IF;
   "Unit1.Em6.ControlNodes".cm.Command.stackTableAxisZ.posAbsolute[0] := #_w1;
END_REGION

REGION Network 250: CmStackTableAxisZ Position Absolute Position1
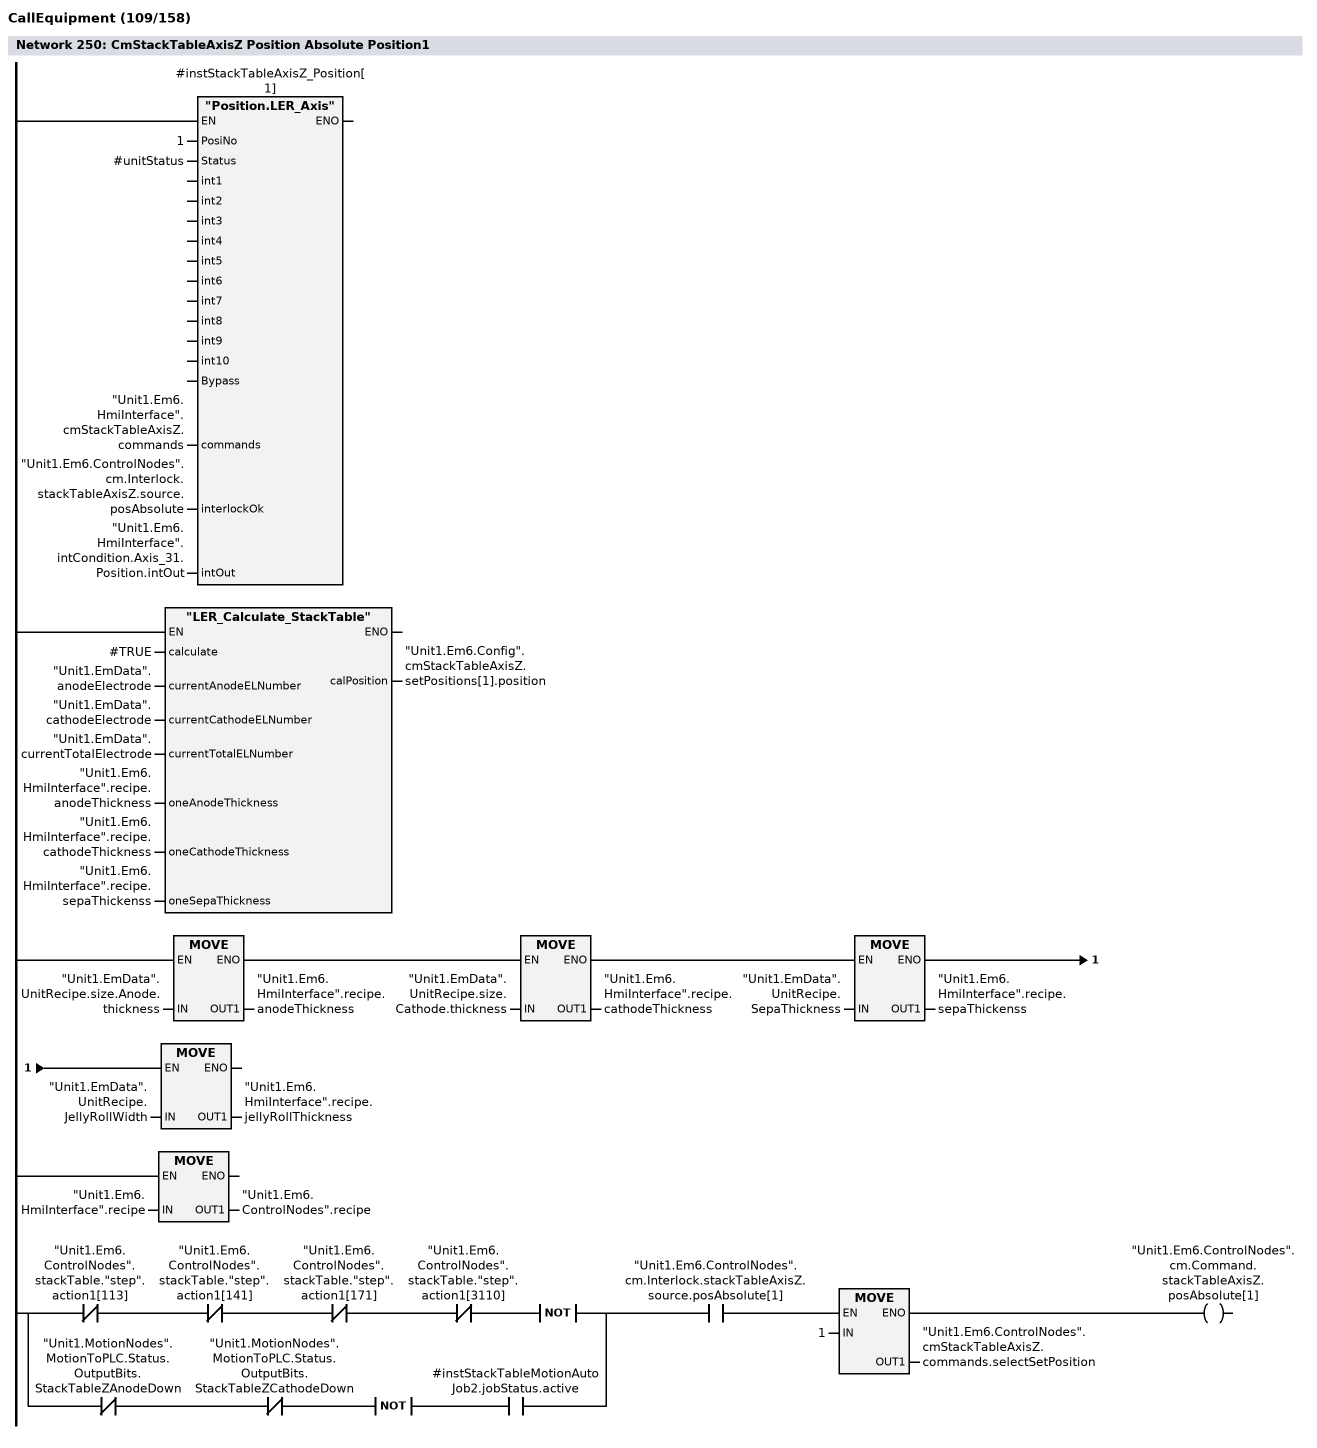
   RUNG wire#powerrail
      #instStackTableAxisZ_Position[1](PosiNo := 1, Status := #unitStatus, int1 :=, int2 :=, int3 :=, int4 :=, int5 :=, int6 :=, int7 :=, int8 :=, int9 :=, int10 :=, Bypass :=, commands := "Unit1.Em6.HmiInterface".cmStackTableAxisZ.commands, interlockOk := "Unit1.Em6.ControlNodes".cm.Interlock.stackTableAxisZ.source.posAbsolute, intOut := "Unit1.Em6.HmiInterface".intCondition.Axis_31.Position.intOut)
   END_RUNG
   RUNG wire#powerrail
      "LER_Calculate_StackTable"(calculate := #TRUE, currentAnodeELNumber := "Unit1.EmData".anodeElectrode, currentCathodeELNumber := "Unit1.EmData".cathodeElectrode, currentTotalELNumber := "Unit1.EmData".currentTotalElectrode, oneAnodeThickness := "Unit1.Em6.HmiInterface".recipe.anodeThickness, oneCathodeThickness := "Unit1.Em6.HmiInterface".recipe.cathodeThickness, oneSepaThickness := "Unit1.Em6.HmiInterface".recipe.sepaThickenss, calPosition => "Unit1.Em6.Config".cmStackTableAxisZ.setPositions[1].position)
   END_RUNG
   RUNG wire#powerrail
      Move(in := "Unit1.EmData".UnitRecipe.size.Anode.thickness, out1 => "Unit1.Em6.HmiInterface".recipe.anodeThickness)
      Move(in := "Unit1.EmData".UnitRecipe.size.Cathode.thickness, out1 => "Unit1.Em6.HmiInterface".recipe.cathodeThickness)
      Move(in := "Unit1.EmData".UnitRecipe.SepaThickness, out1 => "Unit1.Em6.HmiInterface".recipe.sepaThickenss)
      Move(in := "Unit1.EmData".UnitRecipe.JellyRollWidth, out1 => "Unit1.Em6.HmiInterface".recipe.jellyRollThickness)
   END_RUNG
   RUNG wire#powerrail
      Move(in := "Unit1.Em6.HmiInterface".recipe, out1 => "Unit1.Em6.ControlNodes".recipe)
   END_RUNG
   RUNG wire#powerrail
      I_Contact( "Unit1.Em6.ControlNodes".stackTable."step".action1[113] )
      I_Contact( "Unit1.Em6.ControlNodes".stackTable."step".action1[141] )
      I_Contact( "Unit1.Em6.ControlNodes".stackTable."step".action1[171] )
      I_Contact( "Unit1.Em6.ControlNodes".stackTable."step".action1[3110] )
      Not()
      wire#w1
      Contact( "Unit1.Em6.ControlNodes".cm.Interlock.stackTableAxisZ.source.posAbsolute[1] )
      Move(in := 1, out1 => "Unit1.Em6.ControlNodes".cmStackTableAxisZ.commands.selectSetPosition)
      Coil( "Unit1.Em6.ControlNodes".cm.Command.stackTableAxisZ.posAbsolute[1] )
   END_RUNG
   RUNG wire#powerrail
      I_Contact( "Unit1.MotionNodes".MotionToPLC.Status.OutputBits.StackTableZAnodeDown )
      I_Contact( "Unit1.MotionNodes".MotionToPLC.Status.OutputBits.StackTableZCathodeDown )
      Not()
      Contact( #instStackTableMotionAutoJob2.jobStatus.active )
   END_RUNG wire#w1
   // the same network as SCL:
   #instStackTableAxisZ_Position[1](PosiNo := 1,   // "Position.LER_Axis"
                           Status := #unitStatus,
                           commands := "Unit1.Em6.HmiInterface".cmStackTableAxisZ.commands,
                           interlockOk := "Unit1.Em6.ControlNodes".cm.Interlock.stackTableAxisZ.source.posAbsolute,
                           intOut := "Unit1.Em6.HmiInterface".intCondition.Axis_31.Position.intOut);
   "LER_Calculate_StackTable"(calculate := #TRUE,
                           currentAnodeELNumber := "Unit1.EmData".anodeElectrode,
                           currentCathodeELNumber := "Unit1.EmData".cathodeElectrode,
                           currentTotalELNumber := "Unit1.EmData".currentTotalElectrode,
                           oneAnodeThickness := "Unit1.Em6.HmiInterface".recipe.anodeThickness,
                           oneCathodeThickness := "Unit1.Em6.HmiInterface".recipe.cathodeThickness,
                           oneSepaThickness := "Unit1.Em6.HmiInterface".recipe.sepaThickenss,
                           calPosition => "Unit1.Em6.Config".cmStackTableAxisZ.setPositions[1].position);
   "Unit1.Em6.HmiInterface".recipe.anodeThickness := "Unit1.EmData".UnitRecipe.size.Anode.thickness;
   "Unit1.Em6.HmiInterface".recipe.cathodeThickness := "Unit1.EmData".UnitRecipe.size.Cathode.thickness;
   "Unit1.Em6.HmiInterface".recipe.sepaThickenss := "Unit1.EmData".UnitRecipe.SepaThickness;
   "Unit1.Em6.HmiInterface".recipe.jellyRollThickness := "Unit1.EmData".UnitRecipe.JellyRollWidth;
   "Unit1.Em6.ControlNodes".recipe := "Unit1.Em6.HmiInterface".recipe;
   #_w1 := (NOT (NOT "Unit1.Em6.ControlNodes".stackTable."step".action1[113] AND NOT "Unit1.Em6.ControlNodes".stackTable."step".action1[141] AND NOT "Unit1.Em6.ControlNodes".stackTable."step".action1[171] AND NOT "Unit1.Em6.ControlNodes".stackTable."step".action1[3110]) OR (NOT (NOT "Unit1.MotionNodes".MotionToPLC.Status.OutputBits.StackTableZAnodeDown AND NOT "Unit1.MotionNodes".MotionToPLC.Status.OutputBits.StackTableZCathodeDown) AND #instStackTableMotionAutoJob2.jobStatus.active)) AND "Unit1.Em6.ControlNodes".cm.Interlock.stackTableAxisZ.source.posAbsolute[1];
   IF #_w1 THEN "Unit1.Em6.ControlNodes".cmStackTableAxisZ.commands.selectSetPosition := 1; END_IF;
   "Unit1.Em6.ControlNodes".cm.Command.stackTableAxisZ.posAbsolute[1] := #_w1;
END_REGION

REGION Network 251: CmStackTableAxisZ Position Absolute Position2
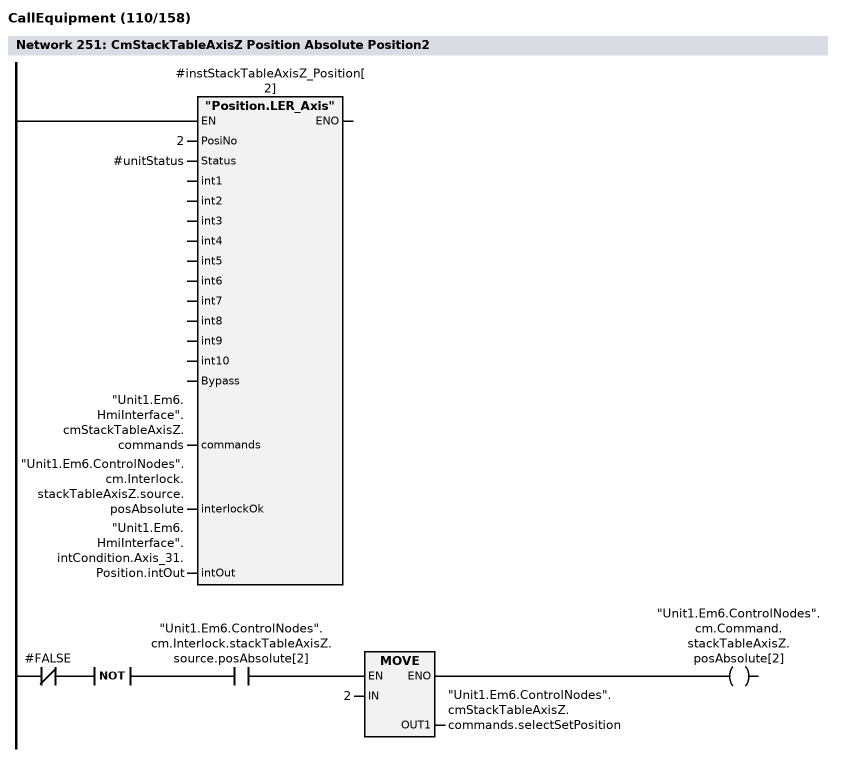
   RUNG wire#powerrail
      #instStackTableAxisZ_Position[2](PosiNo := 2, Status := #unitStatus, int1 :=, int2 :=, int3 :=, int4 :=, int5 :=, int6 :=, int7 :=, int8 :=, int9 :=, int10 :=, Bypass :=, commands := "Unit1.Em6.HmiInterface".cmStackTableAxisZ.commands, interlockOk := "Unit1.Em6.ControlNodes".cm.Interlock.stackTableAxisZ.source.posAbsolute, intOut := "Unit1.Em6.HmiInterface".intCondition.Axis_31.Position.intOut)
   END_RUNG
   RUNG wire#powerrail
      I_Contact( #FALSE )
      Not()
      Contact( "Unit1.Em6.ControlNodes".cm.Interlock.stackTableAxisZ.source.posAbsolute[2] )
      Move(in := 2, out1 => "Unit1.Em6.ControlNodes".cmStackTableAxisZ.commands.selectSetPosition)
      Coil( "Unit1.Em6.ControlNodes".cm.Command.stackTableAxisZ.posAbsolute[2] )
   END_RUNG
   // the same network as SCL:
   #instStackTableAxisZ_Position[2](PosiNo := 2,   // "Position.LER_Axis"
                           Status := #unitStatus,
                           commands := "Unit1.Em6.HmiInterface".cmStackTableAxisZ.commands,
                           interlockOk := "Unit1.Em6.ControlNodes".cm.Interlock.stackTableAxisZ.source.posAbsolute,
                           intOut := "Unit1.Em6.HmiInterface".intCondition.Axis_31.Position.intOut);
   #_w1 := NOT (NOT #FALSE) AND "Unit1.Em6.ControlNodes".cm.Interlock.stackTableAxisZ.source.posAbsolute[2];
   IF #_w1 THEN "Unit1.Em6.ControlNodes".cmStackTableAxisZ.commands.selectSetPosition := 2; END_IF;
   "Unit1.Em6.ControlNodes".cm.Command.stackTableAxisZ.posAbsolute[2] := #_w1;
END_REGION

REGION Network 252: CmStackTableAxisZ Position Absolute Position3
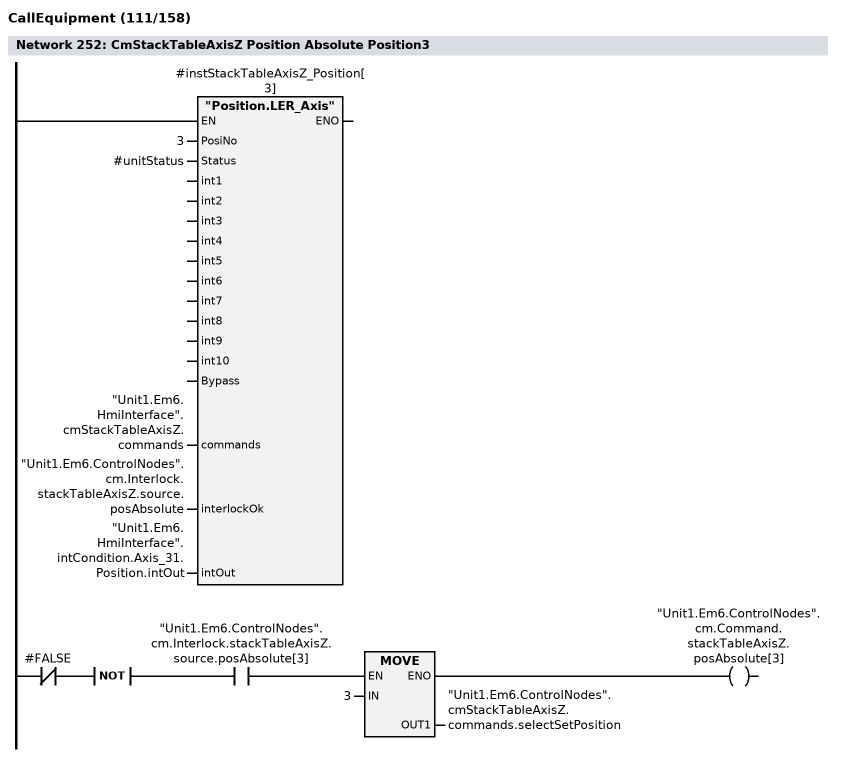
   RUNG wire#powerrail
      #instStackTableAxisZ_Position[3](PosiNo := 3, Status := #unitStatus, int1 :=, int2 :=, int3 :=, int4 :=, int5 :=, int6 :=, int7 :=, int8 :=, int9 :=, int10 :=, Bypass :=, commands := "Unit1.Em6.HmiInterface".cmStackTableAxisZ.commands, interlockOk := "Unit1.Em6.ControlNodes".cm.Interlock.stackTableAxisZ.source.posAbsolute, intOut := "Unit1.Em6.HmiInterface".intCondition.Axis_31.Position.intOut)
   END_RUNG
   RUNG wire#powerrail
      I_Contact( #FALSE )
      Not()
      Contact( "Unit1.Em6.ControlNodes".cm.Interlock.stackTableAxisZ.source.posAbsolute[3] )
      Move(in := 3, out1 => "Unit1.Em6.ControlNodes".cmStackTableAxisZ.commands.selectSetPosition)
      Coil( "Unit1.Em6.ControlNodes".cm.Command.stackTableAxisZ.posAbsolute[3] )
   END_RUNG
   // the same network as SCL:
   #instStackTableAxisZ_Position[3](PosiNo := 3,   // "Position.LER_Axis"
                           Status := #unitStatus,
                           commands := "Unit1.Em6.HmiInterface".cmStackTableAxisZ.commands,
                           interlockOk := "Unit1.Em6.ControlNodes".cm.Interlock.stackTableAxisZ.source.posAbsolute,
                           intOut := "Unit1.Em6.HmiInterface".intCondition.Axis_31.Position.intOut);
   #_w1 := NOT (NOT #FALSE) AND "Unit1.Em6.ControlNodes".cm.Interlock.stackTableAxisZ.source.posAbsolute[3];
   IF #_w1 THEN "Unit1.Em6.ControlNodes".cmStackTableAxisZ.commands.selectSetPosition := 3; END_IF;
   "Unit1.Em6.ControlNodes".cm.Command.stackTableAxisZ.posAbsolute[3] := #_w1;
END_REGION

REGION Network 253: CmStackTableAxisZ Position Absolute Position4
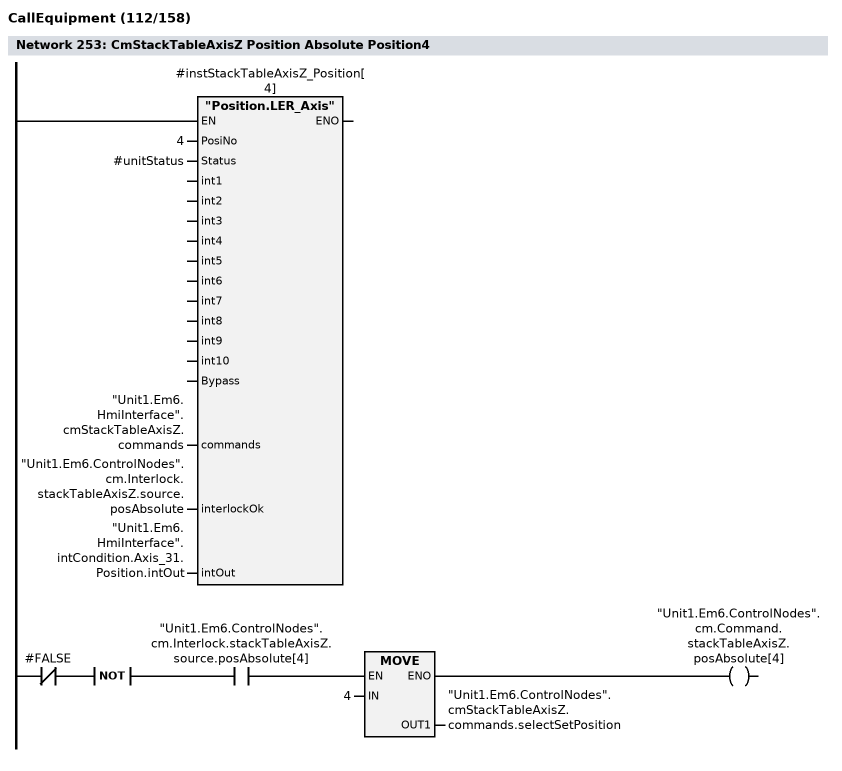
   RUNG wire#powerrail
      #instStackTableAxisZ_Position[4](PosiNo := 4, Status := #unitStatus, int1 :=, int2 :=, int3 :=, int4 :=, int5 :=, int6 :=, int7 :=, int8 :=, int9 :=, int10 :=, Bypass :=, commands := "Unit1.Em6.HmiInterface".cmStackTableAxisZ.commands, interlockOk := "Unit1.Em6.ControlNodes".cm.Interlock.stackTableAxisZ.source.posAbsolute, intOut := "Unit1.Em6.HmiInterface".intCondition.Axis_31.Position.intOut)
   END_RUNG
   RUNG wire#powerrail
      I_Contact( #FALSE )
      Not()
      Contact( "Unit1.Em6.ControlNodes".cm.Interlock.stackTableAxisZ.source.posAbsolute[4] )
      Move(in := 4, out1 => "Unit1.Em6.ControlNodes".cmStackTableAxisZ.commands.selectSetPosition)
      Coil( "Unit1.Em6.ControlNodes".cm.Command.stackTableAxisZ.posAbsolute[4] )
   END_RUNG
   // the same network as SCL:
   #instStackTableAxisZ_Position[4](PosiNo := 4,   // "Position.LER_Axis"
                           Status := #unitStatus,
                           commands := "Unit1.Em6.HmiInterface".cmStackTableAxisZ.commands,
                           interlockOk := "Unit1.Em6.ControlNodes".cm.Interlock.stackTableAxisZ.source.posAbsolute,
                           intOut := "Unit1.Em6.HmiInterface".intCondition.Axis_31.Position.intOut);
   #_w1 := NOT (NOT #FALSE) AND "Unit1.Em6.ControlNodes".cm.Interlock.stackTableAxisZ.source.posAbsolute[4];
   IF #_w1 THEN "Unit1.Em6.ControlNodes".cmStackTableAxisZ.commands.selectSetPosition := 4; END_IF;
   "Unit1.Em6.ControlNodes".cm.Command.stackTableAxisZ.posAbsolute[4] := #_w1;
END_REGION

REGION Network 254: CmStackTableAxisZ Position Absolute Position5
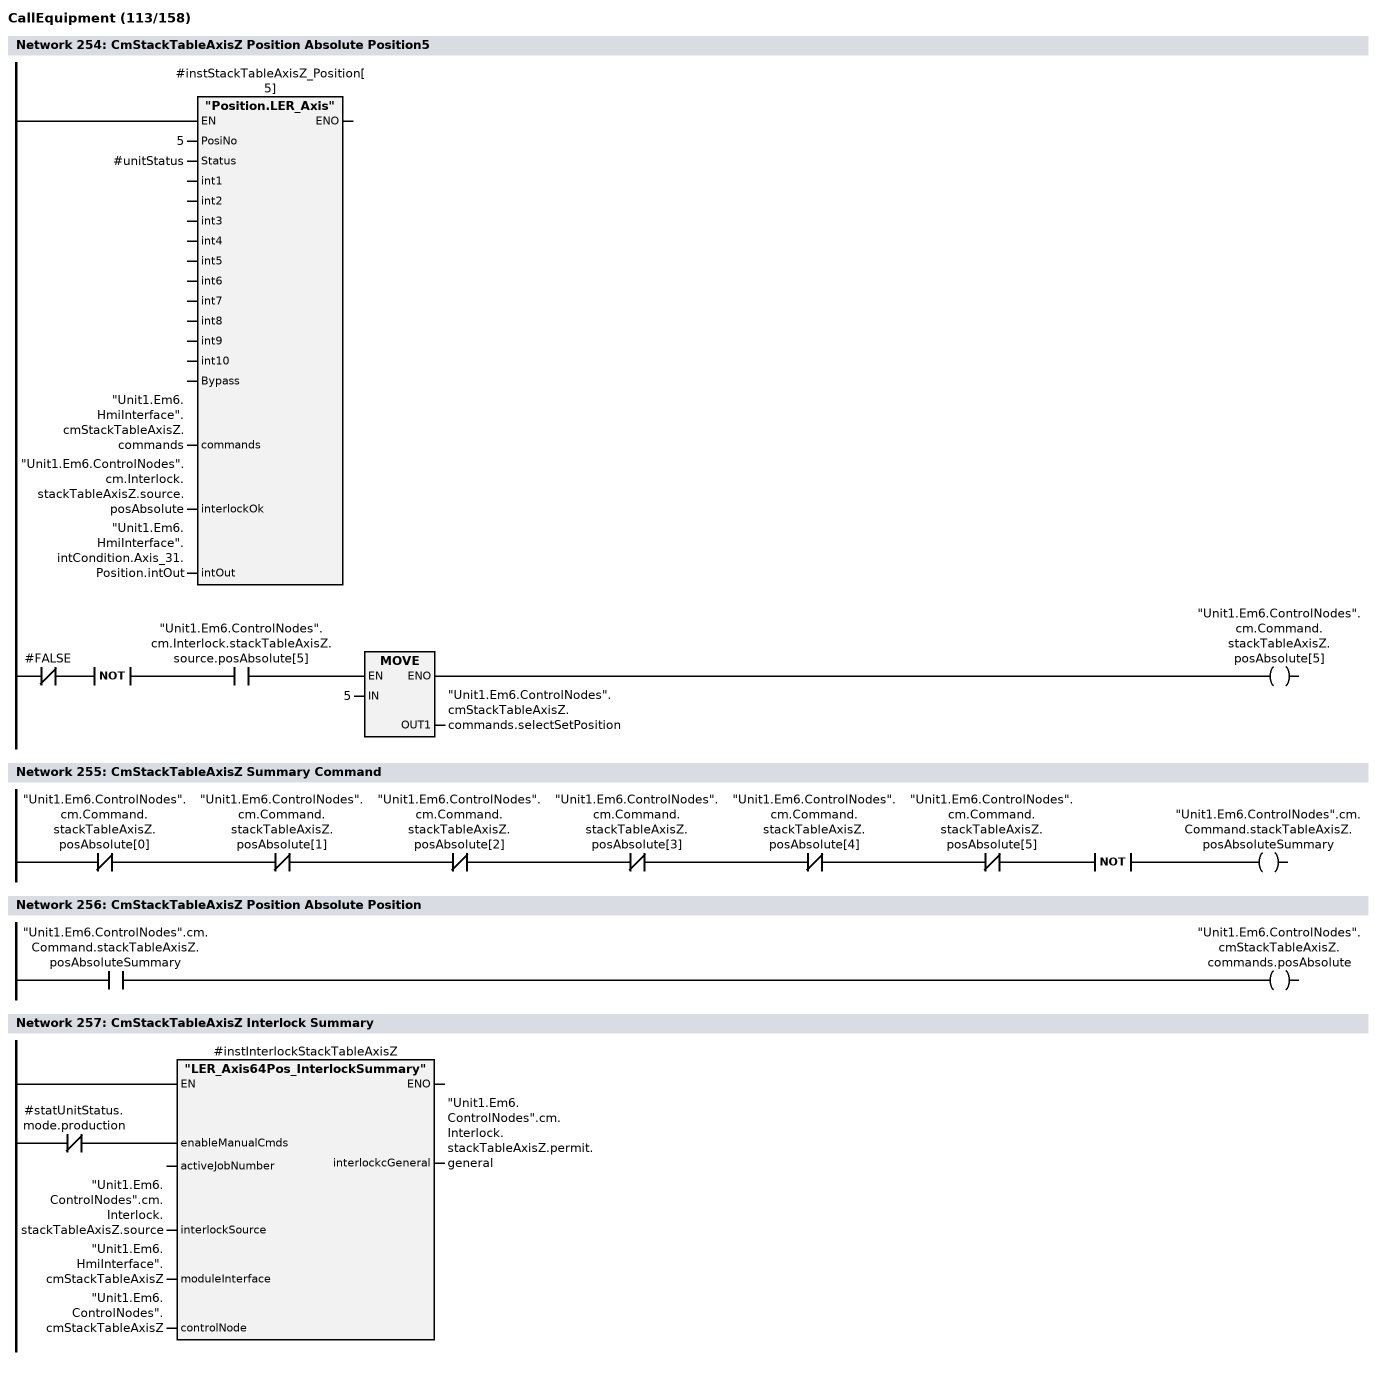
   RUNG wire#powerrail
      #instStackTableAxisZ_Position[5](PosiNo := 5, Status := #unitStatus, int1 :=, int2 :=, int3 :=, int4 :=, int5 :=, int6 :=, int7 :=, int8 :=, int9 :=, int10 :=, Bypass :=, commands := "Unit1.Em6.HmiInterface".cmStackTableAxisZ.commands, interlockOk := "Unit1.Em6.ControlNodes".cm.Interlock.stackTableAxisZ.source.posAbsolute, intOut := "Unit1.Em6.HmiInterface".intCondition.Axis_31.Position.intOut)
   END_RUNG
   RUNG wire#powerrail
      I_Contact( #FALSE )
      Not()
      Contact( "Unit1.Em6.ControlNodes".cm.Interlock.stackTableAxisZ.source.posAbsolute[5] )
      Move(in := 5, out1 => "Unit1.Em6.ControlNodes".cmStackTableAxisZ.commands.selectSetPosition)
      Coil( "Unit1.Em6.ControlNodes".cm.Command.stackTableAxisZ.posAbsolute[5] )
   END_RUNG
   // the same network as SCL:
   #instStackTableAxisZ_Position[5](PosiNo := 5,   // "Position.LER_Axis"
                           Status := #unitStatus,
                           commands := "Unit1.Em6.HmiInterface".cmStackTableAxisZ.commands,
                           interlockOk := "Unit1.Em6.ControlNodes".cm.Interlock.stackTableAxisZ.source.posAbsolute,
                           intOut := "Unit1.Em6.HmiInterface".intCondition.Axis_31.Position.intOut);
   #_w1 := NOT (NOT #FALSE) AND "Unit1.Em6.ControlNodes".cm.Interlock.stackTableAxisZ.source.posAbsolute[5];
   IF #_w1 THEN "Unit1.Em6.ControlNodes".cmStackTableAxisZ.commands.selectSetPosition := 5; END_IF;
   "Unit1.Em6.ControlNodes".cm.Command.stackTableAxisZ.posAbsolute[5] := #_w1;
END_REGION

REGION Network 255: CmStackTableAxisZ Summary Command
   RUNG wire#powerrail
      I_Contact( "Unit1.Em6.ControlNodes".cm.Command.stackTableAxisZ.posAbsolute[0] )
      I_Contact( "Unit1.Em6.ControlNodes".cm.Command.stackTableAxisZ.posAbsolute[1] )
      I_Contact( "Unit1.Em6.ControlNodes".cm.Command.stackTableAxisZ.posAbsolute[2] )
      I_Contact( "Unit1.Em6.ControlNodes".cm.Command.stackTableAxisZ.posAbsolute[3] )
      I_Contact( "Unit1.Em6.ControlNodes".cm.Command.stackTableAxisZ.posAbsolute[4] )
      I_Contact( "Unit1.Em6.ControlNodes".cm.Command.stackTableAxisZ.posAbsolute[5] )
      Not()
      Coil( "Unit1.Em6.ControlNodes".cm.Command.stackTableAxisZ.posAbsoluteSummary )
   END_RUNG
   // the same network as SCL:
   "Unit1.Em6.ControlNodes".cm.Command.stackTableAxisZ.posAbsoluteSummary := NOT (NOT "Unit1.Em6.ControlNodes".cm.Command.stackTableAxisZ.posAbsolute[0] AND NOT "Unit1.Em6.ControlNodes".cm.Command.stackTableAxisZ.posAbsolute[1] AND NOT "Unit1.Em6.ControlNodes".cm.Command.stackTableAxisZ.posAbsolute[2] AND NOT "Unit1.Em6.ControlNodes".cm.Command.stackTableAxisZ.posAbsolute[3] AND NOT "Unit1.Em6.ControlNodes".cm.Command.stackTableAxisZ.posAbsolute[4] AND NOT "Unit1.Em6.ControlNodes".cm.Command.stackTableAxisZ.posAbsolute[5]);
END_REGION

REGION Network 256: CmStackTableAxisZ Position Absolute Position
   RUNG wire#powerrail
      Contact( "Unit1.Em6.ControlNodes".cm.Command.stackTableAxisZ.posAbsoluteSummary )
      Coil( "Unit1.Em6.ControlNodes".cmStackTableAxisZ.commands.posAbsolute )
   END_RUNG
   // the same network as SCL:
   "Unit1.Em6.ControlNodes".cmStackTableAxisZ.commands.posAbsolute := "Unit1.Em6.ControlNodes".cm.Command.stackTableAxisZ.posAbsoluteSummary;
END_REGION

REGION Network 257: CmStackTableAxisZ Interlock Summary
   RUNG wire#powerrail
      #instInterlockStackTableAxisZ(enableManualCmds := wire#w1, activeJobNumber :=, interlockSource := "Unit1.Em6.ControlNodes".cm.Interlock.stackTableAxisZ.source, moduleInterface := "Unit1.Em6.HmiInterface".cmStackTableAxisZ, controlNode := "Unit1.Em6.ControlNodes".cmStackTableAxisZ, interlockcGeneral => "Unit1.Em6.ControlNodes".cm.Interlock.stackTableAxisZ.permit.general)
   END_RUNG
   RUNG wire#powerrail
      I_Contact( #statUnitStatus.mode.production )
   END_RUNG wire#w1
   // the same network as SCL:
   #instInterlockStackTableAxisZ(enableManualCmds := NOT #statUnitStatus.mode.production,   // "LER_Axis64Pos_InterlockSummary"
                           interlockSource := "Unit1.Em6.ControlNodes".cm.Interlock.stackTableAxisZ.source,
                           moduleInterface := "Unit1.Em6.HmiInterface".cmStackTableAxisZ,
                           controlNode := "Unit1.Em6.ControlNodes".cmStackTableAxisZ,
                           interlockcGeneral => "Unit1.Em6.ControlNodes".cm.Interlock.stackTableAxisZ.permit.general);
END_REGION

REGION Network 258: CmStackTableAxisZ velocity/speed
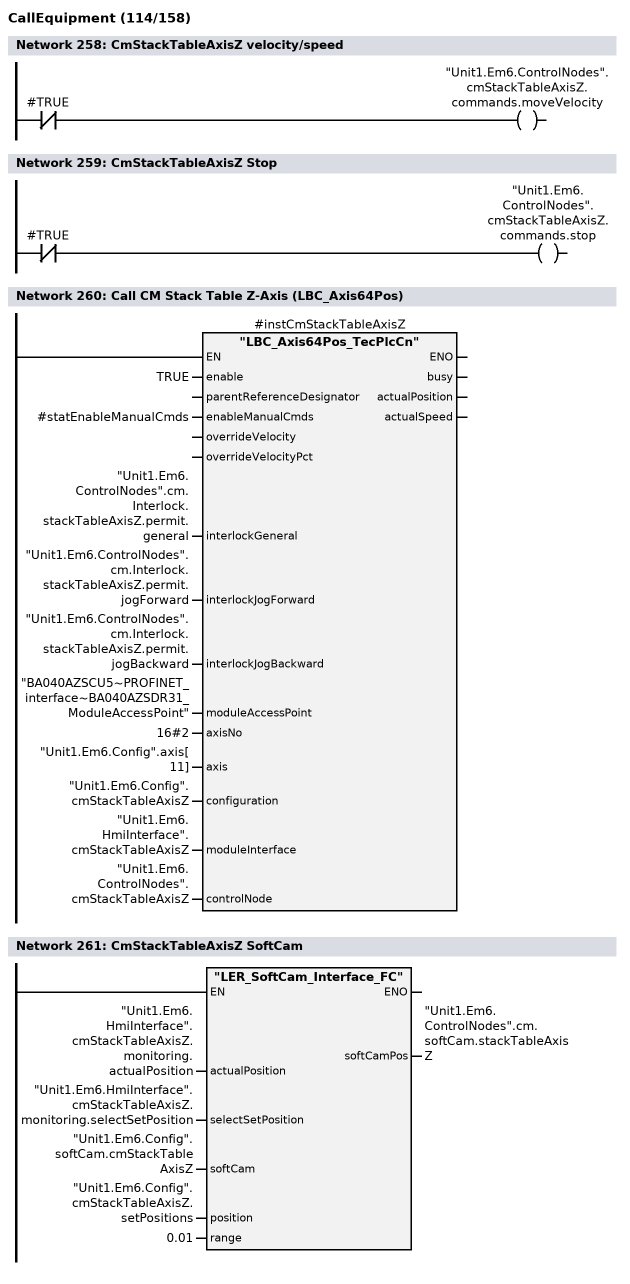
   RUNG wire#powerrail
      I_Contact( #TRUE )
      Coil( "Unit1.Em6.ControlNodes".cmStackTableAxisZ.commands.moveVelocity )
   END_RUNG
   // the same network as SCL:
   "Unit1.Em6.ControlNodes".cmStackTableAxisZ.commands.moveVelocity := NOT #TRUE;
END_REGION

REGION Network 259: CmStackTableAxisZ Stop
   RUNG wire#powerrail
      I_Contact( #TRUE )
      Coil( "Unit1.Em6.ControlNodes".cmStackTableAxisZ.commands.stop )
   END_RUNG
   // the same network as SCL:
   "Unit1.Em6.ControlNodes".cmStackTableAxisZ.commands.stop := NOT #TRUE;
END_REGION

REGION Network 260: Call CM Stack Table Z-Axis (LBC_Axis64Pos)
   RUNG wire#powerrail
      #instCmStackTableAxisZ(enable := TRUE, parentReferenceDesignator :=, enableManualCmds := #statEnableManualCmds, overrideVelocity :=, overrideVelocityPct :=, interlockGeneral := "Unit1.Em6.ControlNodes".cm.Interlock.stackTableAxisZ.permit.general, interlockJogForward := "Unit1.Em6.ControlNodes".cm.Interlock.stackTableAxisZ.permit.jogForward, interlockJogBackward := "Unit1.Em6.ControlNodes".cm.Interlock.stackTableAxisZ.permit.jogBackward, moduleAccessPoint := "BA040AZSCU5~PROFINET_interface~BA040AZSDR31_ModuleAccessPoint", axisNo := 16#2, axis := "Unit1.Em6.Config".axis[11], configuration := "Unit1.Em6.Config".cmStackTableAxisZ, moduleInterface := "Unit1.Em6.HmiInterface".cmStackTableAxisZ, controlNode := "Unit1.Em6.ControlNodes".cmStackTableAxisZ, busy =>, actualPosition =>, actualSpeed =>)
   END_RUNG
   // the same network as SCL:
   #instCmStackTableAxisZ(enable := TRUE,   // "LBC_Axis64Pos_TecPlcCn"
                          enableManualCmds := #statEnableManualCmds,
                          interlockGeneral := "Unit1.Em6.ControlNodes".cm.Interlock.stackTableAxisZ.permit.general,
                          interlockJogForward := "Unit1.Em6.ControlNodes".cm.Interlock.stackTableAxisZ.permit.jogForward,
                          interlockJogBackward := "Unit1.Em6.ControlNodes".cm.Interlock.stackTableAxisZ.permit.jogBackward,
                          moduleAccessPoint := "BA040AZSCU5~PROFINET_interface~BA040AZSDR31_ModuleAccessPoint",
                          axisNo := 16#2,
                          axis := "Unit1.Em6.Config".axis[11],
                          configuration := "Unit1.Em6.Config".cmStackTableAxisZ,
                          moduleInterface := "Unit1.Em6.HmiInterface".cmStackTableAxisZ,
                          controlNode := "Unit1.Em6.ControlNodes".cmStackTableAxisZ);
END_REGION

REGION Network 261: CmStackTableAxisZ SoftCam
   RUNG wire#powerrail
      "LER_SoftCam_Interface_FC"(actualPosition := "Unit1.Em6.HmiInterface".cmStackTableAxisZ.monitoring.actualPosition, selectSetPosition := "Unit1.Em6.HmiInterface".cmStackTableAxisZ.monitoring.selectSetPosition, softCam := "Unit1.Em6.Config".softCam.cmStackTableAxisZ, position := "Unit1.Em6.Config".cmStackTableAxisZ.setPositions, range := 0.01, softCamPos => "Unit1.Em6.ControlNodes".cm.softCam.stackTableAxisZ)
   END_RUNG
   // the same network as SCL:
   "LER_SoftCam_Interface_FC"(actualPosition := "Unit1.Em6.HmiInterface".cmStackTableAxisZ.monitoring.actualPosition,
                           selectSetPosition := "Unit1.Em6.HmiInterface".cmStackTableAxisZ.monitoring.selectSetPosition,
                           softCam := "Unit1.Em6.Config".softCam.cmStackTableAxisZ,
                           position := "Unit1.Em6.Config".cmStackTableAxisZ.setPositions,
                           range := 0.01,
                           softCamPos => "Unit1.Em6.ControlNodes".cm.softCam.stackTableAxisZ);
END_REGION

REGION Network 263: StackTableOutFrontAxisZ Enable
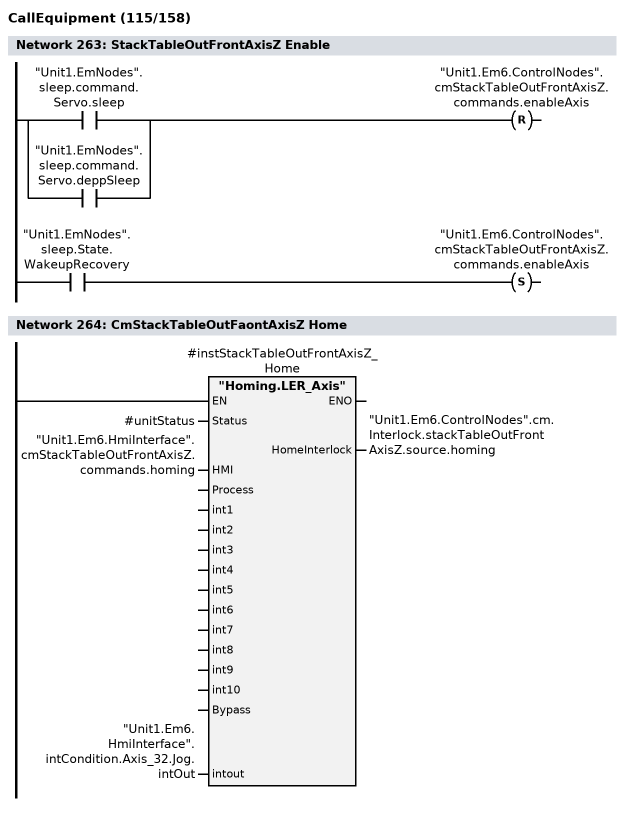
   RUNG wire#powerrail
      Contact( "Unit1.EmNodes".sleep.command.Servo.sleep )
      wire#w1
      R_Coil( "Unit1.Em6.ControlNodes".cmStackTableOutFrontAxisZ.commands.enableAxis )
   END_RUNG
   RUNG wire#powerrail
      Contact( "Unit1.EmNodes".sleep.command.Servo.deppSleep )
   END_RUNG wire#w1
   RUNG wire#powerrail
      Contact( "Unit1.EmNodes".sleep.State.WakeupRecovery )
      S_Coil( "Unit1.Em6.ControlNodes".cmStackTableOutFrontAxisZ.commands.enableAxis )
   END_RUNG
   // the same network as SCL:
   IF "Unit1.EmNodes".sleep.command.Servo.sleep OR "Unit1.EmNodes".sleep.command.Servo.deppSleep THEN
       "Unit1.Em6.ControlNodes".cmStackTableOutFrontAxisZ.commands.enableAxis := FALSE;
   END_IF;
   IF "Unit1.EmNodes".sleep.State.WakeupRecovery THEN
       "Unit1.Em6.ControlNodes".cmStackTableOutFrontAxisZ.commands.enableAxis := TRUE;
   END_IF;
END_REGION

REGION Network 264: CmStackTableOutFaontAxisZ Home
   RUNG wire#powerrail
      #instStackTableOutFrontAxisZ_Home(Status := #unitStatus, HMI := "Unit1.Em6.HmiInterface".cmStackTableOutFrontAxisZ.commands.homing, Process :=, int1 :=, int2 :=, int3 :=, int4 :=, int5 :=, int6 :=, int7 :=, int8 :=, int9 :=, int10 :=, Bypass :=, intout := "Unit1.Em6.HmiInterface".intCondition.Axis_32.Jog.intOut, HomeInterlock => "Unit1.Em6.ControlNodes".cm.Interlock.stackTableOutFrontAxisZ.source.homing)
   END_RUNG
   // the same network as SCL:
   #instStackTableOutFrontAxisZ_Home(Status := #unitStatus,   // "Homing.LER_Axis"
                           HMI := "Unit1.Em6.HmiInterface".cmStackTableOutFrontAxisZ.commands.homing,
                           intout := "Unit1.Em6.HmiInterface".intCondition.Axis_32.Jog.intOut,
                           HomeInterlock => "Unit1.Em6.ControlNodes".cm.Interlock.stackTableOutFrontAxisZ.source.homing);
END_REGION

REGION Network 265: CmStackTableOutFrontAxisZ Position Absolute Jog
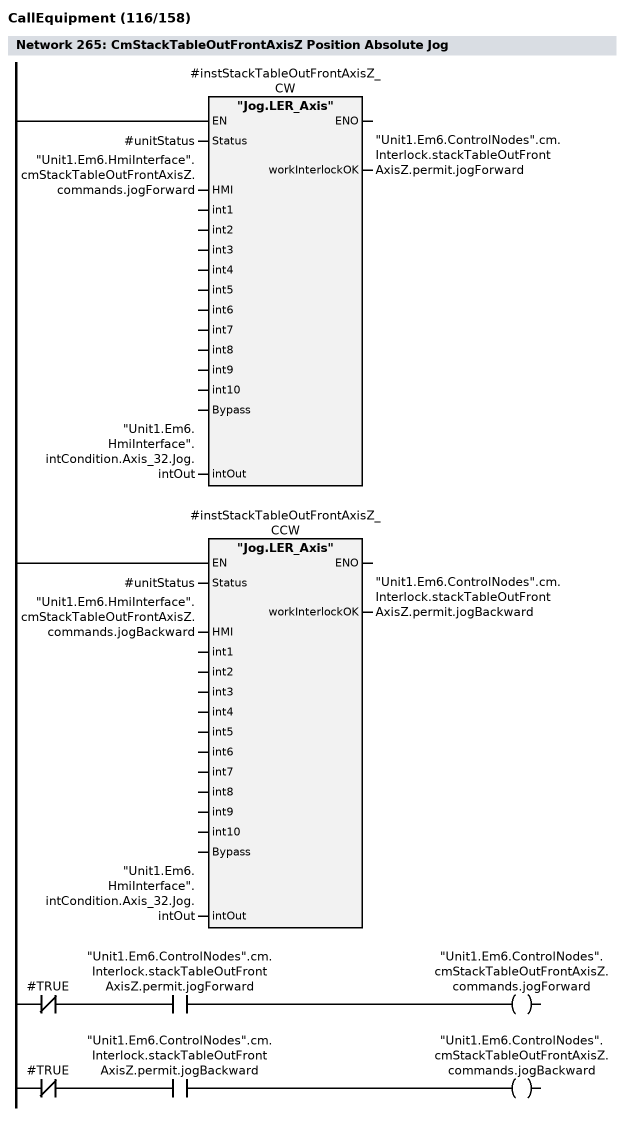
   RUNG wire#powerrail
      #instStackTableOutFrontAxisZ_CW(Status := #unitStatus, HMI := "Unit1.Em6.HmiInterface".cmStackTableOutFrontAxisZ.commands.jogForward, int1 :=, int2 :=, int3 :=, int4 :=, int5 :=, int6 :=, int7 :=, int8 :=, int9 :=, int10 :=, Bypass :=, intOut := "Unit1.Em6.HmiInterface".intCondition.Axis_32.Jog.intOut, workInterlockOK => "Unit1.Em6.ControlNodes".cm.Interlock.stackTableOutFrontAxisZ.permit.jogForward)
   END_RUNG
   RUNG wire#powerrail
      #instStackTableOutFrontAxisZ_CCW(Status := #unitStatus, HMI := "Unit1.Em6.HmiInterface".cmStackTableOutFrontAxisZ.commands.jogBackward, int1 :=, int2 :=, int3 :=, int4 :=, int5 :=, int6 :=, int7 :=, int8 :=, int9 :=, int10 :=, Bypass :=, intOut := "Unit1.Em6.HmiInterface".intCondition.Axis_32.Jog.intOut, workInterlockOK => "Unit1.Em6.ControlNodes".cm.Interlock.stackTableOutFrontAxisZ.permit.jogBackward)
   END_RUNG
   RUNG wire#powerrail
      I_Contact( #TRUE )
      Contact( "Unit1.Em6.ControlNodes".cm.Interlock.stackTableOutFrontAxisZ.permit.jogForward )
      Coil( "Unit1.Em6.ControlNodes".cmStackTableOutFrontAxisZ.commands.jogForward )
   END_RUNG
   RUNG wire#powerrail
      I_Contact( #TRUE )
      Contact( "Unit1.Em6.ControlNodes".cm.Interlock.stackTableOutFrontAxisZ.permit.jogBackward )
      Coil( "Unit1.Em6.ControlNodes".cmStackTableOutFrontAxisZ.commands.jogBackward )
   END_RUNG
   // the same network as SCL:
   #instStackTableOutFrontAxisZ_CW(Status := #unitStatus,   // "Jog.LER_Axis"
                           HMI := "Unit1.Em6.HmiInterface".cmStackTableOutFrontAxisZ.commands.jogForward,
                           intOut := "Unit1.Em6.HmiInterface".intCondition.Axis_32.Jog.intOut,
                           workInterlockOK => "Unit1.Em6.ControlNodes".cm.Interlock.stackTableOutFrontAxisZ.permit.jogForward);
   #instStackTableOutFrontAxisZ_CCW(Status := #unitStatus,   // "Jog.LER_Axis"
                           HMI := "Unit1.Em6.HmiInterface".cmStackTableOutFrontAxisZ.commands.jogBackward,
                           intOut := "Unit1.Em6.HmiInterface".intCondition.Axis_32.Jog.intOut,
                           workInterlockOK => "Unit1.Em6.ControlNodes".cm.Interlock.stackTableOutFrontAxisZ.permit.jogBackward);
   "Unit1.Em6.ControlNodes".cmStackTableOutFrontAxisZ.commands.jogForward := NOT #TRUE AND "Unit1.Em6.ControlNodes".cm.Interlock.stackTableOutFrontAxisZ.permit.jogForward;
   "Unit1.Em6.ControlNodes".cmStackTableOutFrontAxisZ.commands.jogBackward := NOT #TRUE AND "Unit1.Em6.ControlNodes".cm.Interlock.stackTableOutFrontAxisZ.permit.jogBackward;
END_REGION

REGION Network 266: CmStackTableOutFrontAxisZ Position Absolute Position0
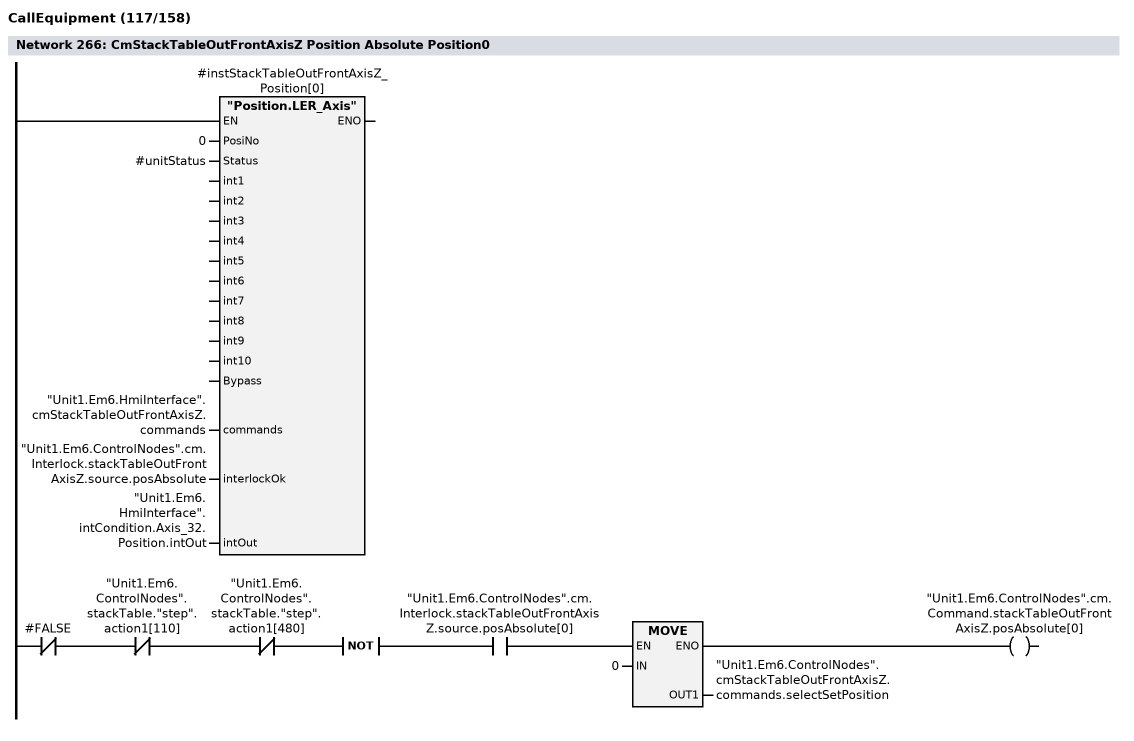
   RUNG wire#powerrail
      #instStackTableOutFrontAxisZ_Position[0](PosiNo := 0, Status := #unitStatus, int1 :=, int2 :=, int3 :=, int4 :=, int5 :=, int6 :=, int7 :=, int8 :=, int9 :=, int10 :=, Bypass :=, commands := "Unit1.Em6.HmiInterface".cmStackTableOutFrontAxisZ.commands, interlockOk := "Unit1.Em6.ControlNodes".cm.Interlock.stackTableOutFrontAxisZ.source.posAbsolute, intOut := "Unit1.Em6.HmiInterface".intCondition.Axis_32.Position.intOut)
   END_RUNG
   RUNG wire#powerrail
      I_Contact( #FALSE )
      I_Contact( "Unit1.Em6.ControlNodes".stackTable."step".action1[110] )
      I_Contact( "Unit1.Em6.ControlNodes".stackTable."step".action1[480] )
      Not()
      Contact( "Unit1.Em6.ControlNodes".cm.Interlock.stackTableOutFrontAxisZ.source.posAbsolute[0] )
      Move(in := 0, out1 => "Unit1.Em6.ControlNodes".cmStackTableOutFrontAxisZ.commands.selectSetPosition)
      Coil( "Unit1.Em6.ControlNodes".cm.Command.stackTableOutFrontAxisZ.posAbsolute[0] )
   END_RUNG
   // the same network as SCL:
   #instStackTableOutFrontAxisZ_Position[0](PosiNo := 0,   // "Position.LER_Axis"
                           Status := #unitStatus,
                           commands := "Unit1.Em6.HmiInterface".cmStackTableOutFrontAxisZ.commands,
                           interlockOk := "Unit1.Em6.ControlNodes".cm.Interlock.stackTableOutFrontAxisZ.source.posAbsolute,
                           intOut := "Unit1.Em6.HmiInterface".intCondition.Axis_32.Position.intOut);
   #_w1 := NOT (NOT #FALSE AND NOT "Unit1.Em6.ControlNodes".stackTable."step".action1[110] AND NOT "Unit1.Em6.ControlNodes".stackTable."step".action1[480]) AND "Unit1.Em6.ControlNodes".cm.Interlock.stackTableOutFrontAxisZ.source.posAbsolute[0];
   IF #_w1 THEN "Unit1.Em6.ControlNodes".cmStackTableOutFrontAxisZ.commands.selectSetPosition := 0; END_IF;
   "Unit1.Em6.ControlNodes".cm.Command.stackTableOutFrontAxisZ.posAbsolute[0] := #_w1;
END_REGION

REGION Network 267: CmStackTableOutFrontAxisZ Position Absolute Position1
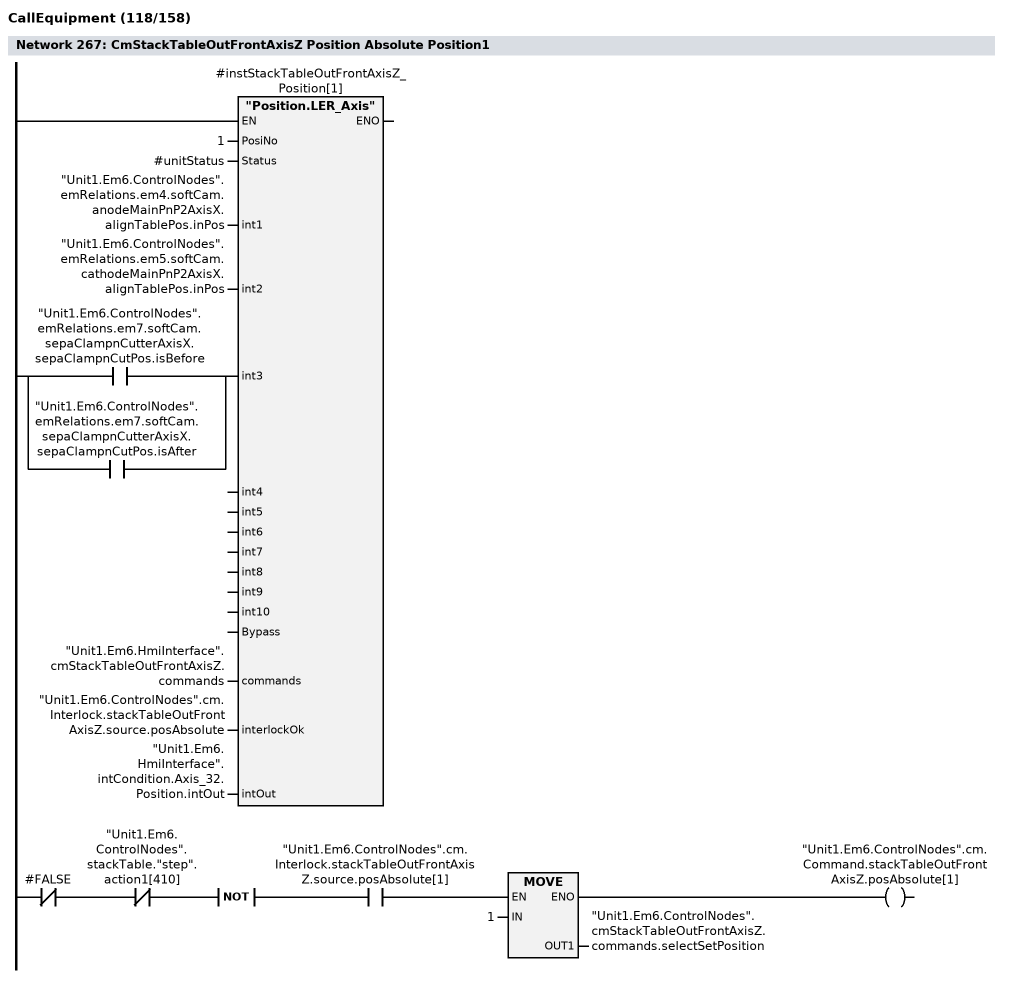
   RUNG wire#powerrail
      #instStackTableOutFrontAxisZ_Position[1](int3 := wire#w1, PosiNo := 1, Status := #unitStatus, int1 := "Unit1.Em6.ControlNodes".emRelations.em4.softCam.anodeMainPnP2AxisX.alignTablePos.inPos, int2 := "Unit1.Em6.ControlNodes".emRelations.em5.softCam.cathodeMainPnP2AxisX.alignTablePos.inPos, int4 :=, int5 :=, int6 :=, int7 :=, int8 :=, int9 :=, int10 :=, Bypass :=, commands := "Unit1.Em6.HmiInterface".cmStackTableOutFrontAxisZ.commands, interlockOk := "Unit1.Em6.ControlNodes".cm.Interlock.stackTableOutFrontAxisZ.source.posAbsolute, intOut := "Unit1.Em6.HmiInterface".intCondition.Axis_32.Position.intOut)
   END_RUNG
   RUNG wire#powerrail
      Contact( "Unit1.Em6.ControlNodes".emRelations.em7.softCam.sepaClampnCutterAxisX.sepaClampnCutPos.isBefore )
   END_RUNG wire#w1
   RUNG wire#powerrail
      Contact( "Unit1.Em6.ControlNodes".emRelations.em7.softCam.sepaClampnCutterAxisX.sepaClampnCutPos.isAfter )
   END_RUNG wire#w1
   RUNG wire#powerrail
      I_Contact( #FALSE )
      I_Contact( "Unit1.Em6.ControlNodes".stackTable."step".action1[410] )
      Not()
      Contact( "Unit1.Em6.ControlNodes".cm.Interlock.stackTableOutFrontAxisZ.source.posAbsolute[1] )
      Move(in := 1, out1 => "Unit1.Em6.ControlNodes".cmStackTableOutFrontAxisZ.commands.selectSetPosition)
      Coil( "Unit1.Em6.ControlNodes".cm.Command.stackTableOutFrontAxisZ.posAbsolute[1] )
   END_RUNG
   // the same network as SCL:
   #instStackTableOutFrontAxisZ_Position[1](PosiNo := 1,   // "Position.LER_Axis"
                           Status := #unitStatus,
                           int1 := "Unit1.Em6.ControlNodes".emRelations.em4.softCam.anodeMainPnP2AxisX.alignTablePos.inPos,
                           int2 := "Unit1.Em6.ControlNodes".emRelations.em5.softCam.cathodeMainPnP2AxisX.alignTablePos.inPos,
                           int3 := "Unit1.Em6.ControlNodes".emRelations.em7.softCam.sepaClampnCutterAxisX.sepaClampnCutPos.isBefore OR "Unit1.Em6.ControlNodes".emRelations.em7.softCam.sepaClampnCutterAxisX.sepaClampnCutPos.isAfter,
                           commands := "Unit1.Em6.HmiInterface".cmStackTableOutFrontAxisZ.commands,
                           interlockOk := "Unit1.Em6.ControlNodes".cm.Interlock.stackTableOutFrontAxisZ.source.posAbsolute,
                           intOut := "Unit1.Em6.HmiInterface".intCondition.Axis_32.Position.intOut);
   #_w1 := NOT (NOT #FALSE AND NOT "Unit1.Em6.ControlNodes".stackTable."step".action1[410]) AND "Unit1.Em6.ControlNodes".cm.Interlock.stackTableOutFrontAxisZ.source.posAbsolute[1];
   IF #_w1 THEN "Unit1.Em6.ControlNodes".cmStackTableOutFrontAxisZ.commands.selectSetPosition := 1; END_IF;
   "Unit1.Em6.ControlNodes".cm.Command.stackTableOutFrontAxisZ.posAbsolute[1] := #_w1;
END_REGION

REGION Network 268: CmStackTableOutFrontAxisZ Position Absolute Position2
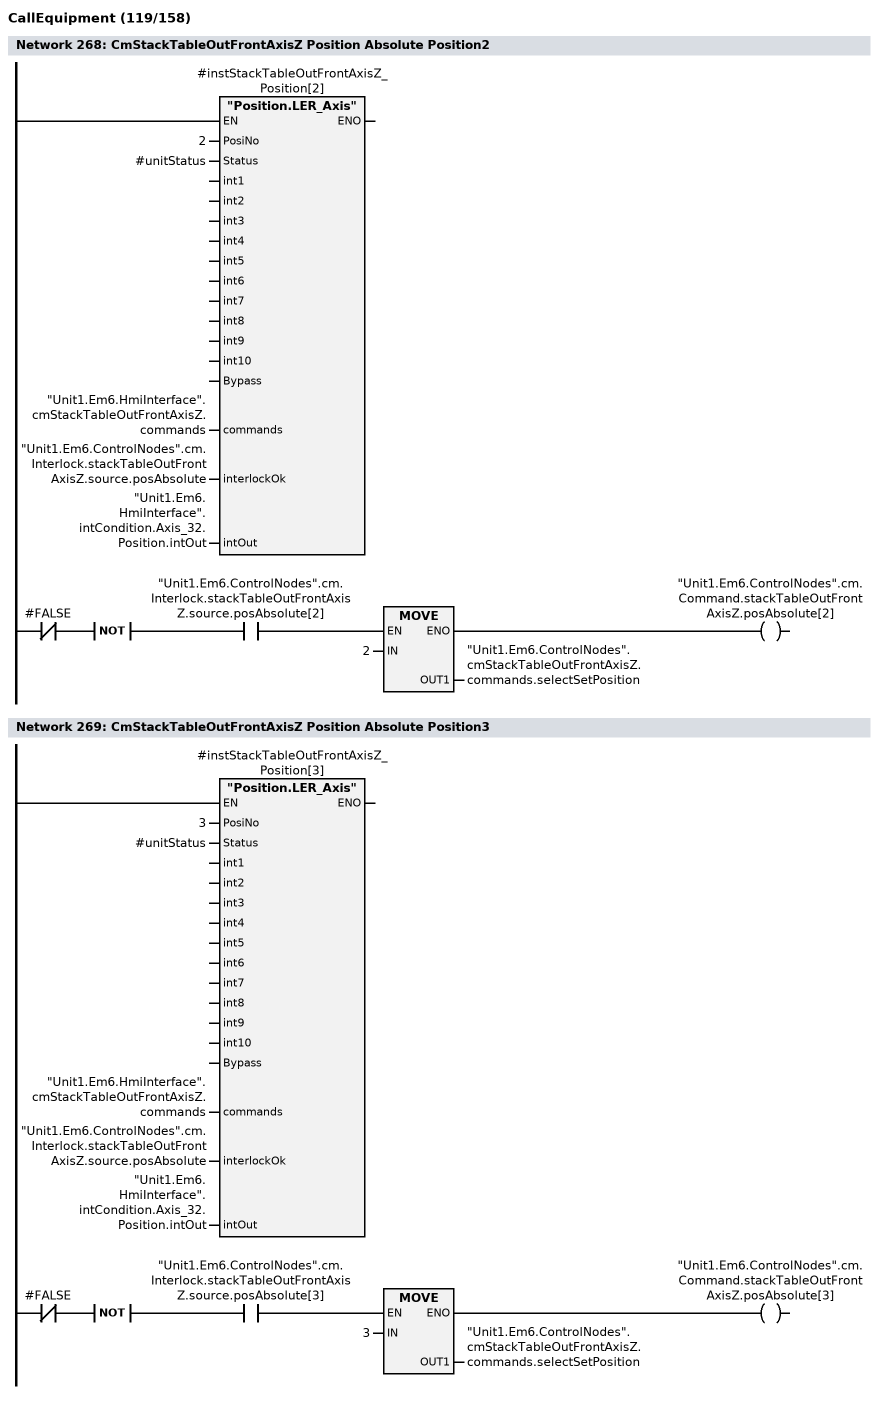
   RUNG wire#powerrail
      #instStackTableOutFrontAxisZ_Position[2](PosiNo := 2, Status := #unitStatus, int1 :=, int2 :=, int3 :=, int4 :=, int5 :=, int6 :=, int7 :=, int8 :=, int9 :=, int10 :=, Bypass :=, commands := "Unit1.Em6.HmiInterface".cmStackTableOutFrontAxisZ.commands, interlockOk := "Unit1.Em6.ControlNodes".cm.Interlock.stackTableOutFrontAxisZ.source.posAbsolute, intOut := "Unit1.Em6.HmiInterface".intCondition.Axis_32.Position.intOut)
   END_RUNG
   RUNG wire#powerrail
      I_Contact( #FALSE )
      Not()
      Contact( "Unit1.Em6.ControlNodes".cm.Interlock.stackTableOutFrontAxisZ.source.posAbsolute[2] )
      Move(in := 2, out1 => "Unit1.Em6.ControlNodes".cmStackTableOutFrontAxisZ.commands.selectSetPosition)
      Coil( "Unit1.Em6.ControlNodes".cm.Command.stackTableOutFrontAxisZ.posAbsolute[2] )
   END_RUNG
   // the same network as SCL:
   #instStackTableOutFrontAxisZ_Position[2](PosiNo := 2,   // "Position.LER_Axis"
                           Status := #unitStatus,
                           commands := "Unit1.Em6.HmiInterface".cmStackTableOutFrontAxisZ.commands,
                           interlockOk := "Unit1.Em6.ControlNodes".cm.Interlock.stackTableOutFrontAxisZ.source.posAbsolute,
                           intOut := "Unit1.Em6.HmiInterface".intCondition.Axis_32.Position.intOut);
   #_w1 := NOT (NOT #FALSE) AND "Unit1.Em6.ControlNodes".cm.Interlock.stackTableOutFrontAxisZ.source.posAbsolute[2];
   IF #_w1 THEN "Unit1.Em6.ControlNodes".cmStackTableOutFrontAxisZ.commands.selectSetPosition := 2; END_IF;
   "Unit1.Em6.ControlNodes".cm.Command.stackTableOutFrontAxisZ.posAbsolute[2] := #_w1;
END_REGION

REGION Network 269: CmStackTableOutFrontAxisZ Position Absolute Position3
   RUNG wire#powerrail
      #instStackTableOutFrontAxisZ_Position[3](PosiNo := 3, Status := #unitStatus, int1 :=, int2 :=, int3 :=, int4 :=, int5 :=, int6 :=, int7 :=, int8 :=, int9 :=, int10 :=, Bypass :=, commands := "Unit1.Em6.HmiInterface".cmStackTableOutFrontAxisZ.commands, interlockOk := "Unit1.Em6.ControlNodes".cm.Interlock.stackTableOutFrontAxisZ.source.posAbsolute, intOut := "Unit1.Em6.HmiInterface".intCondition.Axis_32.Position.intOut)
   END_RUNG
   RUNG wire#powerrail
      I_Contact( #FALSE )
      Not()
      Contact( "Unit1.Em6.ControlNodes".cm.Interlock.stackTableOutFrontAxisZ.source.posAbsolute[3] )
      Move(in := 3, out1 => "Unit1.Em6.ControlNodes".cmStackTableOutFrontAxisZ.commands.selectSetPosition)
      Coil( "Unit1.Em6.ControlNodes".cm.Command.stackTableOutFrontAxisZ.posAbsolute[3] )
   END_RUNG
   // the same network as SCL:
   #instStackTableOutFrontAxisZ_Position[3](PosiNo := 3,   // "Position.LER_Axis"
                           Status := #unitStatus,
                           commands := "Unit1.Em6.HmiInterface".cmStackTableOutFrontAxisZ.commands,
                           interlockOk := "Unit1.Em6.ControlNodes".cm.Interlock.stackTableOutFrontAxisZ.source.posAbsolute,
                           intOut := "Unit1.Em6.HmiInterface".intCondition.Axis_32.Position.intOut);
   #_w1 := NOT (NOT #FALSE) AND "Unit1.Em6.ControlNodes".cm.Interlock.stackTableOutFrontAxisZ.source.posAbsolute[3];
   IF #_w1 THEN "Unit1.Em6.ControlNodes".cmStackTableOutFrontAxisZ.commands.selectSetPosition := 3; END_IF;
   "Unit1.Em6.ControlNodes".cm.Command.stackTableOutFrontAxisZ.posAbsolute[3] := #_w1;
END_REGION

REGION Network 270: CmStackTableOutFrontAxisZ Position Absolute Position4
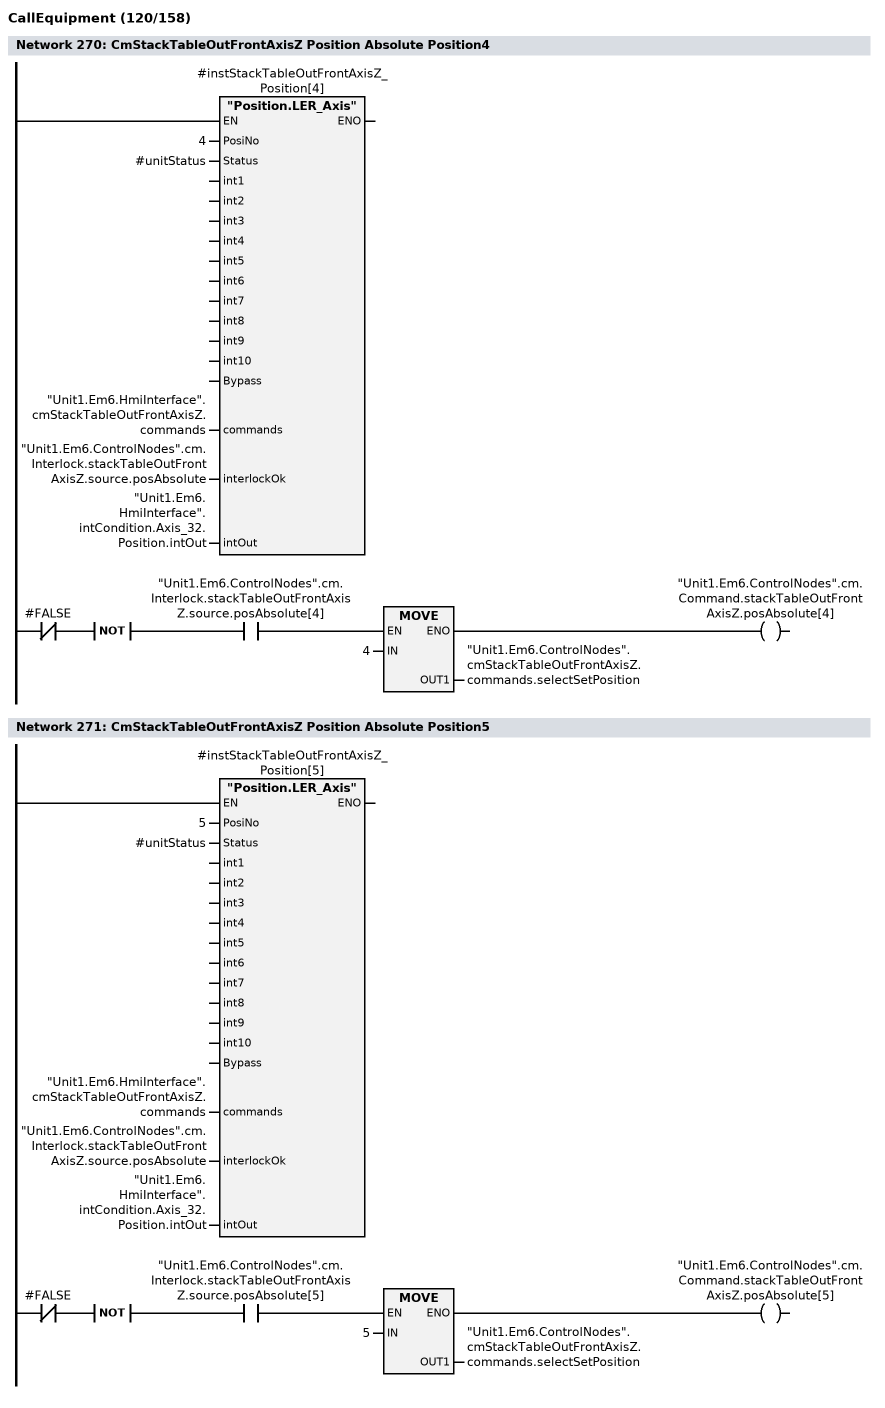
   RUNG wire#powerrail
      #instStackTableOutFrontAxisZ_Position[4](PosiNo := 4, Status := #unitStatus, int1 :=, int2 :=, int3 :=, int4 :=, int5 :=, int6 :=, int7 :=, int8 :=, int9 :=, int10 :=, Bypass :=, commands := "Unit1.Em6.HmiInterface".cmStackTableOutFrontAxisZ.commands, interlockOk := "Unit1.Em6.ControlNodes".cm.Interlock.stackTableOutFrontAxisZ.source.posAbsolute, intOut := "Unit1.Em6.HmiInterface".intCondition.Axis_32.Position.intOut)
   END_RUNG
   RUNG wire#powerrail
      I_Contact( #FALSE )
      Not()
      Contact( "Unit1.Em6.ControlNodes".cm.Interlock.stackTableOutFrontAxisZ.source.posAbsolute[4] )
      Move(in := 4, out1 => "Unit1.Em6.ControlNodes".cmStackTableOutFrontAxisZ.commands.selectSetPosition)
      Coil( "Unit1.Em6.ControlNodes".cm.Command.stackTableOutFrontAxisZ.posAbsolute[4] )
   END_RUNG
   // the same network as SCL:
   #instStackTableOutFrontAxisZ_Position[4](PosiNo := 4,   // "Position.LER_Axis"
                           Status := #unitStatus,
                           commands := "Unit1.Em6.HmiInterface".cmStackTableOutFrontAxisZ.commands,
                           interlockOk := "Unit1.Em6.ControlNodes".cm.Interlock.stackTableOutFrontAxisZ.source.posAbsolute,
                           intOut := "Unit1.Em6.HmiInterface".intCondition.Axis_32.Position.intOut);
   #_w1 := NOT (NOT #FALSE) AND "Unit1.Em6.ControlNodes".cm.Interlock.stackTableOutFrontAxisZ.source.posAbsolute[4];
   IF #_w1 THEN "Unit1.Em6.ControlNodes".cmStackTableOutFrontAxisZ.commands.selectSetPosition := 4; END_IF;
   "Unit1.Em6.ControlNodes".cm.Command.stackTableOutFrontAxisZ.posAbsolute[4] := #_w1;
END_REGION

REGION Network 271: CmStackTableOutFrontAxisZ Position Absolute Position5
   RUNG wire#powerrail
      #instStackTableOutFrontAxisZ_Position[5](PosiNo := 5, Status := #unitStatus, int1 :=, int2 :=, int3 :=, int4 :=, int5 :=, int6 :=, int7 :=, int8 :=, int9 :=, int10 :=, Bypass :=, commands := "Unit1.Em6.HmiInterface".cmStackTableOutFrontAxisZ.commands, interlockOk := "Unit1.Em6.ControlNodes".cm.Interlock.stackTableOutFrontAxisZ.source.posAbsolute, intOut := "Unit1.Em6.HmiInterface".intCondition.Axis_32.Position.intOut)
   END_RUNG
   RUNG wire#powerrail
      I_Contact( #FALSE )
      Not()
      Contact( "Unit1.Em6.ControlNodes".cm.Interlock.stackTableOutFrontAxisZ.source.posAbsolute[5] )
      Move(in := 5, out1 => "Unit1.Em6.ControlNodes".cmStackTableOutFrontAxisZ.commands.selectSetPosition)
      Coil( "Unit1.Em6.ControlNodes".cm.Command.stackTableOutFrontAxisZ.posAbsolute[5] )
   END_RUNG
   // the same network as SCL:
   #instStackTableOutFrontAxisZ_Position[5](PosiNo := 5,   // "Position.LER_Axis"
                           Status := #unitStatus,
                           commands := "Unit1.Em6.HmiInterface".cmStackTableOutFrontAxisZ.commands,
                           interlockOk := "Unit1.Em6.ControlNodes".cm.Interlock.stackTableOutFrontAxisZ.source.posAbsolute,
                           intOut := "Unit1.Em6.HmiInterface".intCondition.Axis_32.Position.intOut);
   #_w1 := NOT (NOT #FALSE) AND "Unit1.Em6.ControlNodes".cm.Interlock.stackTableOutFrontAxisZ.source.posAbsolute[5];
   IF #_w1 THEN "Unit1.Em6.ControlNodes".cmStackTableOutFrontAxisZ.commands.selectSetPosition := 5; END_IF;
   "Unit1.Em6.ControlNodes".cm.Command.stackTableOutFrontAxisZ.posAbsolute[5] := #_w1;
END_REGION

REGION Network 272: CmStackTableOutFrontAxisZ Summary Command
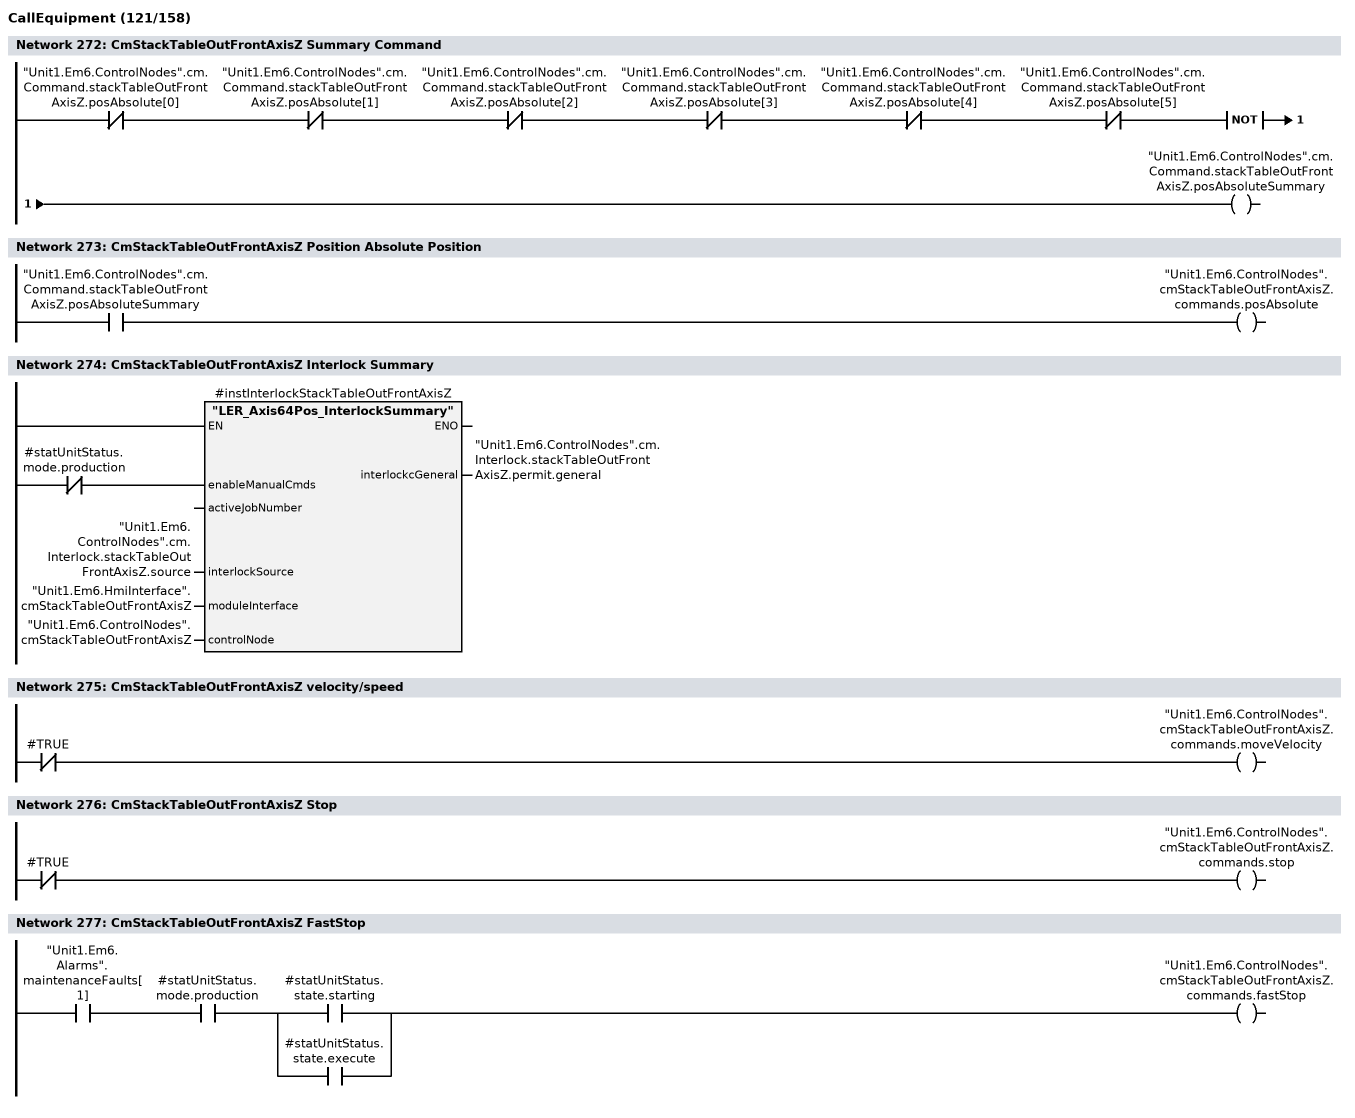
   RUNG wire#powerrail
      I_Contact( "Unit1.Em6.ControlNodes".cm.Command.stackTableOutFrontAxisZ.posAbsolute[0] )
      I_Contact( "Unit1.Em6.ControlNodes".cm.Command.stackTableOutFrontAxisZ.posAbsolute[1] )
      I_Contact( "Unit1.Em6.ControlNodes".cm.Command.stackTableOutFrontAxisZ.posAbsolute[2] )
      I_Contact( "Unit1.Em6.ControlNodes".cm.Command.stackTableOutFrontAxisZ.posAbsolute[3] )
      I_Contact( "Unit1.Em6.ControlNodes".cm.Command.stackTableOutFrontAxisZ.posAbsolute[4] )
      I_Contact( "Unit1.Em6.ControlNodes".cm.Command.stackTableOutFrontAxisZ.posAbsolute[5] )
      Not()
      Coil( "Unit1.Em6.ControlNodes".cm.Command.stackTableOutFrontAxisZ.posAbsoluteSummary )
   END_RUNG
   // the same network as SCL:
   "Unit1.Em6.ControlNodes".cm.Command.stackTableOutFrontAxisZ.posAbsoluteSummary := NOT (NOT "Unit1.Em6.ControlNodes".cm.Command.stackTableOutFrontAxisZ.posAbsolute[0] AND NOT "Unit1.Em6.ControlNodes".cm.Command.stackTableOutFrontAxisZ.posAbsolute[1] AND NOT "Unit1.Em6.ControlNodes".cm.Command.stackTableOutFrontAxisZ.posAbsolute[2] AND NOT "Unit1.Em6.ControlNodes".cm.Command.stackTableOutFrontAxisZ.posAbsolute[3] AND NOT "Unit1.Em6.ControlNodes".cm.Command.stackTableOutFrontAxisZ.posAbsolute[4] AND NOT "Unit1.Em6.ControlNodes".cm.Command.stackTableOutFrontAxisZ.posAbsolute[5]);
END_REGION

REGION Network 273: CmStackTableOutFrontAxisZ Position Absolute Position
   RUNG wire#powerrail
      Contact( "Unit1.Em6.ControlNodes".cm.Command.stackTableOutFrontAxisZ.posAbsoluteSummary )
      Coil( "Unit1.Em6.ControlNodes".cmStackTableOutFrontAxisZ.commands.posAbsolute )
   END_RUNG
   // the same network as SCL:
   "Unit1.Em6.ControlNodes".cmStackTableOutFrontAxisZ.commands.posAbsolute := "Unit1.Em6.ControlNodes".cm.Command.stackTableOutFrontAxisZ.posAbsoluteSummary;
END_REGION

REGION Network 274: CmStackTableOutFrontAxisZ Interlock Summary
   RUNG wire#powerrail
      #instInterlockStackTableOutFrontAxisZ(enableManualCmds := wire#w1, activeJobNumber :=, interlockSource := "Unit1.Em6.ControlNodes".cm.Interlock.stackTableOutFrontAxisZ.source, moduleInterface := "Unit1.Em6.HmiInterface".cmStackTableOutFrontAxisZ, controlNode := "Unit1.Em6.ControlNodes".cmStackTableOutFrontAxisZ, interlockcGeneral => "Unit1.Em6.ControlNodes".cm.Interlock.stackTableOutFrontAxisZ.permit.general)
   END_RUNG
   RUNG wire#powerrail
      I_Contact( #statUnitStatus.mode.production )
   END_RUNG wire#w1
   // the same network as SCL:
   #instInterlockStackTableOutFrontAxisZ(enableManualCmds := NOT #statUnitStatus.mode.production,   // "LER_Axis64Pos_InterlockSummary"
                           interlockSource := "Unit1.Em6.ControlNodes".cm.Interlock.stackTableOutFrontAxisZ.source,
                           moduleInterface := "Unit1.Em6.HmiInterface".cmStackTableOutFrontAxisZ,
                           controlNode := "Unit1.Em6.ControlNodes".cmStackTableOutFrontAxisZ,
                           interlockcGeneral => "Unit1.Em6.ControlNodes".cm.Interlock.stackTableOutFrontAxisZ.permit.general);
END_REGION

REGION Network 275: CmStackTableOutFrontAxisZ velocity/speed
   RUNG wire#powerrail
      I_Contact( #TRUE )
      Coil( "Unit1.Em6.ControlNodes".cmStackTableOutFrontAxisZ.commands.moveVelocity )
   END_RUNG
   // the same network as SCL:
   "Unit1.Em6.ControlNodes".cmStackTableOutFrontAxisZ.commands.moveVelocity := NOT #TRUE;
END_REGION

REGION Network 276: CmStackTableOutFrontAxisZ Stop
   RUNG wire#powerrail
      I_Contact( #TRUE )
      Coil( "Unit1.Em6.ControlNodes".cmStackTableOutFrontAxisZ.commands.stop )
   END_RUNG
   // the same network as SCL:
   "Unit1.Em6.ControlNodes".cmStackTableOutFrontAxisZ.commands.stop := NOT #TRUE;
END_REGION

REGION Network 277: CmStackTableOutFrontAxisZ FastStop
   RUNG wire#powerrail
      Contact( "Unit1.Em6.Alarms".maintenanceFaults[1] )
      Contact( #statUnitStatus.mode.production )
      wire#w1
      Contact( #statUnitStatus.state.starting )
      wire#w2
      Coil( "Unit1.Em6.ControlNodes".cmStackTableOutFrontAxisZ.commands.fastStop )
   END_RUNG
   RUNG wire#w1
      Contact( #statUnitStatus.state.execute )
   END_RUNG wire#w2
   // the same network as SCL:
   "Unit1.Em6.ControlNodes".cmStackTableOutFrontAxisZ.commands.fastStop := "Unit1.Em6.Alarms".maintenanceFaults[1] AND #statUnitStatus.mode.production AND (#statUnitStatus.state.starting OR #statUnitStatus.state.execute);
END_REGION

REGION Network 278: Call CM Stack Table Out Front Z-Axis (LBC_Axis64Pos)
